LIN {X 0,Y 162.399,Z 558.631,A -85,B 0,C 180,E1 -26128.349,E2 -26128.349} C_VEL
LIN {X 0,Y 156.579,Z 567.786,A -85,B 0,C 180,E1 -26130.23,E2 -26130.23} C_VEL
LIN {X 0,Y 150.044,Z 576.728,A -85,B 0,C 180,E1 -26132.532,E2 -26132.532} C_VEL
LIN {X 0,Y 142.728,Z 585.711,A -85,B 0,C 180,E1 -26135.664,E2 -26135.664} C_VEL
LIN {X 0,Y 135.887,Z 593.161,A -85,B 0,C 180,E1 -26139.125,E2 -26139.125} C_VEL
LIN {X 0,Y 129.545,Z 599.346,A -85,B 0,C 180,E1 -26142.914,E2 -26142.914} C_VEL
LIN {X 0,Y 123.734,Z 604.443,A -85,B 0,C 180,E1 -26147.033,E2 -26147.033} C_VEL
LIN {X 0,Y 117.104,Z 609.682,A -85,B 0,C 180,E1 -26153.121,E2 -26153.121} C_VEL
LIN {X 0,Y 111.791,Z 613.372,A -85,B 0,C 180,E1 -26159.806,E2 -26159.806} C_VEL
LIN {X 0,Y 108.032,Z 615.635,A -85,B 0,C 180,E1 -26167.026,E2 -26167.026} C_VEL
LIN {X 0,Y 105.706,Z 616.545,A -85,B 0,C 180,E1 -26174.577,E2 -26174.577} C_VEL
LIN {X 0,Y 105.009,Z 616.121,A -85,B 0,C 180,E1 -26182.308,E2 -26182.308} C_VEL
LIN {X 0,Y 105.077,Z 615.416,A -85,B 0,C 180,E1 -26186.165,E2 -26186.165} C_VEL
LIN {X 0,Y 105.791,Z 613.021,A -85,B 0,C 180,E1 -26193.809,E2 -26193.809} C_VEL
LIN {X 0,Y 107.768,Z 609.248,A -85,B 0,C 180,E1 -26201.282,E2 -26201.282} C_VEL
LIN {X 0,Y 111.163,Z 603.939,A -85,B 0,C 180,E1 -26208.427,E2 -26208.427} C_VEL
LIN {X 0,Y 114.818,Z 598.843,A -85,B 0,C 180,E1 -26213.444,E2 -26213.444} C_VEL
LIN {X 0,Y 119.854,Z 591.564,A -85,B 0,C 180,E1 -26218.931,E2 -26218.931} C_VEL
LIN {X 0,Y 124.817,Z 583.942,A -85,B 0,C 180,E1 -26223.297,E2 -26223.297} C_VEL
LIN {X 0,Y 130.491,Z 574.792,A -85,B 0,C 180,E1 -26227.292,E2 -26227.292} C_VEL
LIN {X 0,Y 136.215,Z 564.684,A -85,B 0,C 180,E1 -26230.645,E2 -26230.645} C_VEL
LIN {X 0,Y 141.727,Z 553.57,A -85,B 0,C 180,E1 -26233.473,E2 -26233.473} C_VEL
LIN {X 0,Y 146.852,Z 541.305,A -85,B 0,C 180,E1 -26235.877,E2 -26235.877} C_VEL
LIN {X 0,Y 151.111,Z 529.497,A -85,B 0,C 180,E1 -26237.587,E2 -26237.587} C_VEL
LIN {X 0,Y 154.843,Z 516.616,A -85,B 0,C 180,E1 -26238.986,E2 -26238.986} C_VEL
LIN {X 0,Y 157.814,Z 502.413,A -85,B 0,C 180,E1 -26240.126,E2 -26240.126} C_VEL
LIN {X 0,Y 159.807,Z 487.984,A -85,B 0,C 180,E1 -26240.867,E2 -26240.867} C_VEL
LIN {X 0,Y 163.436,Z 443.82,A -85,B 0,C 180,E1 -26242.428,E2 -26242.428} C_VEL
LIN {X 0,Y 159.128,Z 434.822,A -85,B 0,C 180,E1 -26245.539,E2 -26245.539} C_VEL
LIN {X 0,Y 155.155,Z 427.48,A -85,B 0,C 180,E1 -26248.763,E2 -26248.763} C_VEL
LIN {X 0,Y 151.706,Z 421.59,A -85,B 0,C 180,E1 -26251.973,E2 -26251.973} C_VEL
LIN {X 0,Y 149.783,Z 418.5,A -85,B 0,C 180,E1 -26253.994,E2 -26253.994} C_VEL
LIN {X 0,Y 147.754,Z 415.273,A -85,B 0,C 180,E1 -26256.389,E2 -26256.389} C_VEL
LIN {X 0,Y 145.207,Z 411.371,A -85,B 0,C 180,E1 -26259.939,E2 -26259.939} C_VEL
LIN {X 0,Y 142.875,Z 408.164,A -85,B 0,C 180,E1 -26264.073,E2 -26264.073} C_VEL
LIN {X 0,Y 142.203,Z 406.763,A -85,B 0,C 180,E1 -26265.692,E2 -26265.692} C_VEL
LIN {X 0,Y 139.978,Z 403.826,A -85,B 0,C 180,E1 -26274.958,E2 -26274.958} C_VEL
LIN {X 0,Y 140.014,Z 403.461,A -85,B 0,C 180,E1 -26278.561,E2 -26278.561} C_VEL
LIN {X 0,Y 140.342,Z 404.521,A -85,B 0,C 180,E1 -26281.793,E2 -26281.793} C_VEL
LIN {X 0,Y 142.46,Z 406.94,A -85,B 0,C 180,E1 -26288.51,E2 -26288.51} C_VEL
LIN {X 0,Y 144.47,Z 410.538,A -85,B 0,C 180,E1 -26292.555,E2 -26292.555} C_VEL
LIN {X 0,Y 145.741,Z 412.18,A -85,B 0,C 180,E1 -26294.508,E2 -26294.508} C_VEL
LIN {X 0,Y 148.649,Z 416.668,A -85,B 0,C 180,E1 -26298.342,E2 -26298.342} C_VEL
LIN {X 0,Y 151.312,Z 420.86,A -85,B 0,C 180,E1 -26301.258,E2 -26301.258} C_VEL
LIN {X 0,Y 154.67,Z 426.429,A -85,B 0,C 180,E1 -26304.431,E2 -26304.431} C_VEL
LIN {X 0,Y 157.563,Z 432.02,A -85,B 0,C 180,E1 -26306.891,E2 -26306.891} C_VEL
LIN {X 0,Y 161.424,Z 442.286,A -85,B 0,C 180,E1 -26310.022,E2 -26310.022} C_VEL
LIN {X 0,Y 163.244,Z 447.912,A -85,B 0,C 180,E1 -26311.422,E2 -26311.422} C_VEL
LIN {X 0,Y 159.088,Z 496.229,A -85,B 0,C 180,E1 -26313.076,E2 -26313.076} C_VEL
LIN {X 0,Y 156.838,Z 510.579,A -85,B 0,C 180,E1 -26313.863,E2 -26313.863} C_VEL
LIN {X 0,Y 153.433,Z 524.942,A -85,B 0,C 180,E1 -26315.041,E2 -26315.041} C_VEL
LIN {X 0,Y 149.545,Z 537.278,A -85,B 0,C 180,E1 -26316.411,E2 -26316.411} C_VEL
LIN {X 0,Y 144.563,Z 550.226,A -85,B 0,C 180,E1 -26318.381,E2 -26318.381} C_VEL
LIN {X 0,Y 139.278,Z 561.994,A -85,B 0,C 180,E1 -26320.81,E2 -26320.81} C_VEL
LIN {X 0,Y 133.684,Z 572.756,A -85,B 0,C 180,E1 -26323.711,E2 -26323.711} C_VEL
LIN {X 0,Y 127.43,Z 583.411,A -85,B 0,C 180,E1 -26327.5,E2 -26327.5} C_VEL
LIN {X 0,Y 121.787,Z 592.198,A -85,B 0,C 180,E1 -26331.659,E2 -26331.659} C_VEL
LIN {X 0,Y 116.209,Z 600.631,A -85,B 0,C 180,E1 -26337.025,E2 -26337.025} C_VEL
LIN {X 0,Y 112.275,Z 606.497,A -85,B 0,C 180,E1 -26342.001,E2 -26342.001} C_VEL
LIN {X 0,Y 109.209,Z 611.326,A -85,B 0,C 180,E1 -26347.287,E2 -26347.287} C_VEL
LIN {X 0,Y 106.398,Z 616.311,A -85,B 0,C 180,E1 -26354.68,E2 -26354.68} C_VEL
LIN {X 0,Y 105.166,Z 619.78,A -85,B 0,C 180,E1 -26362.319,E2 -26362.319} C_VEL
LIN {X 0,Y 105.166,Z 621.827,A -85,B 0,C 180,E1 -26370,E2 -26370} C_VEL
LIN {X 0,Y 105.195,Z 622.477,A -85,B 0,C 180,E1 -26377.679,E2 -26377.679} C_VEL
LIN {X 0,Y 106.498,Z 621.795,A -85,B 0,C 180,E1 -26385.305,E2 -26385.305} C_VEL
LIN {X 0,Y 109.463,Z 619.789,A -85,B 0,C 180,E1 -26392.657,E2 -26392.657} C_VEL
LIN {X 0,Y 114.037,Z 616.407,A -85,B 0,C 180,E1 -26399.539,E2 -26399.539} C_VEL
LIN {X 0,Y 118.372,Z 612.921,A -85,B 0,C 180,E1 -26404.334,E2 -26404.334} C_VEL
LIN {X 0,Y 121.014,Z 610.729,A -85,B 0,C 180,E1 -26406.692,E2 -26406.692} C_VEL
LIN {X 0,Y 123.209,Z 608.466,A -85,B 0,C 180,E1 -26409.042,E2 -26409.042} C_VEL
LIN {X 0,Y 125.615,Z 604.474,A -85,B 0,C 180,E1 -26413.085,E2 -26413.085} C_VEL
LIN {X 0,Y 128.462,Z 599.904,A -85,B 0,C 180,E1 -26416.838,E2 -26416.838} C_VEL
LIN {X 0,Y 131.222,Z 596.74,A -85,B 0,C 180,E1 -26418.667,E2 -26418.667} C_VEL
LIN {X 0,Y 139.696,Z 587.753,A -85,B 0,C 180,E1 -26422.406,E2 -26422.406} C_VEL
LIN {X 0,Y 147.43,Z 578.268,A -85,B 0,C 180,E1 -26425.314,E2 -26425.314} C_VEL
LIN {X 0,Y 154.898,Z 567.778,A -85,B 0,C 180,E1 -26427.675,E2 -26427.675} C_VEL
LIN {X 0,Y 161.912,Z 556.21,A -85,B 0,C 180,E1 -26429.618,E2 -26429.618} C_VEL
LIN {X 0,Y 168.417,Z 543.379,A -85,B 0,C 180,E1 -26431.199,E2 -26431.199} C_VEL
LIN {X 0,Y 173.581,Z 530.831,A -85,B 0,C 180,E1 -26432.332,E2 -26432.332} C_VEL
LIN {X 0,Y 177.858,Z 517.413,A -85,B 0,C 180,E1 -26433.247,E2 -26433.247} C_VEL
LIN {X 0,Y 181.081,Z 503.535,A -85,B 0,C 180,E1 -26433.906,E2 -26433.906} C_VEL
LIN {X 0,Y 183.19,Z 488.883,A -85,B 0,C 180,E1 -26434.353,E2 -26434.353} C_VEL
LIN {X 0,Y 184.85,Z 471.444,A -85,B 0,C 180,E1 -26434.848,E2 -26434.848} C_VEL
LIN {X 0,Y 182.027,Z 462.8,A -85,B 0,C 180,E1 -26438.096,E2 -26438.096} C_VEL
LIN {X 0,Y 179.629,Z 456.499,A -85,B 0,C 180,E1 -26441.299,E2 -26441.299} C_VEL
LIN {X 0,Y 177.45,Z 452.505,A -85,B 0,C 180,E1 -26444.685,E2 -26444.685} C_VEL
LIN {X 0,Y 175.833,Z 449.251,A -85,B 0,C 180,E1 -26448.107,E2 -26448.107} C_VEL
LIN {X 0,Y 174.341,Z 445.787,A -85,B 0,C 180,E1 -26453.782,E2 -26453.782} C_VEL
LIN {X 0,Y 174.27,Z 445.225,A -85,B 0,C 180,E1 -26454.656,E2 -26454.656} C_VEL
LIN {X 0,Y 174.337,Z 445.109,A -85,B 0,C 180,E1 -26460.145,E2 -26460.145} C_VEL
LIN {X 0,Y 175.732,Z 448.882,A -85,B 0,C 180,E1 -26466.027,E2 -26466.027} C_VEL
LIN {X 0,Y 176.557,Z 450.738,A -85,B 0,C 180,E1 -26468.009,E2 -26468.009} C_VEL
LIN {X 0,Y 178.07,Z 453.628,A -85,B 0,C 180,E1 -26470.806,E2 -26470.806} C_VEL
LIN {X 0,Y 180.172,Z 457.72,A -85,B 0,C 180,E1 -26473.896,E2 -26473.896} C_VEL
LIN {X 0,Y 182.541,Z 462.521,A -85,B 0,C 180,E1 -26476.766,E2 -26476.766} C_VEL
LIN {X 0,Y 185.162,Z 468.275,A -85,B 0,C 180,E1 -26479.506,E2 -26479.506} C_VEL
LIN {X 0,Y 182.433,Z 493.552,A -85,B 0,C 180,E1 -26480.188,E2 -26480.188} C_VEL
LIN {X 0,Y 179.908,Z 506.993,A -85,B 0,C 180,E1 -26480.783,E2 -26480.783} C_VEL
LIN {X 0,Y 176.286,Z 520.463,A -85,B 0,C 180,E1 -26481.662,E2 -26481.662} C_VEL
LIN {X 0,Y 171.504,Z 533.661,A -85,B 0,C 180,E1 -26482.781,E2 -26482.781} C_VEL
LIN {X 0,Y 165.72,Z 546.39,A -85,B 0,C 180,E1 -26484.25,E2 -26484.25} C_VEL
LIN {X 0,Y 159.25,Z 558.074,A -85,B 0,C 180,E1 -26486.026,E2 -26486.026} C_VEL
LIN {X 0,Y 153.016,Z 567.649,A -85,B 0,C 180,E1 -26487.923,E2 -26487.923} C_VEL
LIN {X 0,Y 146.289,Z 576.569,A -85,B 0,C 180,E1 -26490.148,E2 -26490.148} C_VEL
LIN {X 0,Y 138.639,Z 585.613,A -85,B 0,C 180,E1 -26493.237,E2 -26493.237} C_VEL
LIN {X 0,Y 131.447,Z 593.117,A -85,B 0,C 180,E1 -26496.681,E2 -26496.681} C_VEL
LIN {X 0,Y 124.728,Z 599.348,A -85,B 0,C 180,E1 -26500.478,E2 -26500.478} C_VEL
LIN {X 0,Y 118.558,Z 604.472,A -85,B 0,C 180,E1 -26504.657,E2 -26504.657} C_VEL
LIN {X 0,Y 113.05,Z 608.576,A -85,B 0,C 180,E1 -26509.252,E2 -26509.252} C_VEL
LIN {X 0,Y 108.302,Z 611.817,A -85,B 0,C 180,E1 -26514.266,E2 -26514.266} C_VEL
LIN {X 0,Y 103.348,Z 614.818,A -85,B 0,C 180,E1 -26521.575,E2 -26521.575} C_VEL
LIN {X 0,Y 99.921,Z 616.434,A -85,B 0,C 180,E1 -26529.411,E2 -26529.411} C_VEL
LIN {X 0,Y 98.157,Z 616.711,A -85,B 0,C 180,E1 -26537.597,E2 -26537.597} C_VEL
LIN {X 0,Y 97.916,Z 616.351,A -85,B 0,C 180,E1 -26541.747,E2 -26541.747} C_VEL
LIN {X 0,Y 97.955,Z 615.663,A -85,B 0,C 180,E1 -26545.886,E2 -26545.886} C_VEL
LIN {X 0,Y 98.489,Z 613.862,A -85,B 0,C 180,E1 -26552.507,E2 -26552.507} C_VEL
LIN {X 0,Y 100.145,Z 610.623,A -85,B 0,C 180,E1 -26560.104,E2 -26560.104} C_VEL
LIN {X 0,Y 103.446,Z 605.748,A -85,B 0,C 180,E1 -26567.801,E2 -26567.801} C_VEL
LIN {X 0,Y 108.372,Z 599.241,A -85,B 0,C 180,E1 -26574.93,E2 -26574.93} C_VEL
LIN {X 0,Y 113.705,Z 592.01,A -85,B 0,C 180,E1 -26580.658,E2 -26580.658} C_VEL
LIN {X 0,Y 119.932,Z 583.053,A -85,B 0,C 180,E1 -26585.872,E2 -26585.872} C_VEL
LIN {X 0,Y 126.016,Z 573.655,A -85,B 0,C 180,E1 -26589.892,E2 -26589.892} C_VEL
LIN {X 0,Y 132.065,Z 563.253,A -85,B 0,C 180,E1 -26593.246,E2 -26593.246} C_VEL
LIN {X 0,Y 137.885,Z 551.772,A -85,B 0,C 180,E1 -26596.049,E2 -26596.049} C_VEL
LIN {X 0,Y 143.246,Z 539.058,A -85,B 0,C 180,E1 -26598.433,E2 -26598.433} C_VEL
LIN {X 0,Y 147.711,Z 526.619,A -85,B 0,C 180,E1 -26600.103,E2 -26600.103} C_VEL
LIN {X 0,Y 151.593,Z 512.787,A -85,B 0,C 180,E1 -26601.473,E2 -26601.473} C_VEL
LIN {X 0,Y 154.383,Z 498.867,A -85,B 0,C 180,E1 -26602.453,E2 -26602.453} C_VEL
LIN {X 0,Y 156.03,Z 485.645,A -85,B 0,C 180,E1 -26603.065,E2 -26603.065} C_VEL
LIN {X 0,Y 159.29,Z 446.776,A -85,B 0,C 180,E1 -26604.439,E2 -26604.439} C_VEL
LIN {X 0,Y 155.497,Z 438.74,A -85,B 0,C 180,E1 -26607.464,E2 -26607.464} C_VEL
LIN {X 0,Y 151.515,Z 431.095,A -85,B 0,C 180,E1 -26611.088,E2 -26611.088} C_VEL
LIN {X 0,Y 147.933,Z 424.893,A -85,B 0,C 180,E1 -26614.934,E2 -26614.934} C_VEL
LIN {X 0,Y 145.849,Z 421.5,A -85,B 0,C 180,E1 -26617.575,E2 -26617.575} C_VEL
LIN {X 0,Y 143.612,Z 417.914,A -85,B 0,C 180,E1 -26620.965,E2 -26620.965} C_VEL
LIN {X 0,Y 141.494,Z 414.599,A -85,B 0,C 180,E1 -26625.141,E2 -26625.141} C_VEL
LIN {X 0,Y 140.971,Z 413.609,A -85,B 0,C 180,E1 -26626.496,E2 -26626.496} C_VEL
LIN {X 0,Y 139.081,Z 410.76,A -85,B 0,C 180,E1 -26635.652,E2 -26635.652} C_VEL
LIN {X 0,Y 139.161,Z 410.509,A -85,B 0,C 180,E1 -26638.748,E2 -26638.748} C_VEL
LIN {X 0,Y 141.212,Z 413.663,A -85,B 0,C 180,E1 -26647.686,E2 -26647.686} C_VEL
LIN {X 0,Y 143.208,Z 417.38,A -85,B 0,C 180,E1 -26651.993,E2 -26651.993} C_VEL
LIN {X 0,Y 144.165,Z 418.711,A -85,B 0,C 180,E1 -26653.568,E2 -26653.568} C_VEL
LIN {X 0,Y 146.863,Z 423.102,A -85,B 0,C 180,E1 -26657.391,E2 -26657.391} C_VEL
LIN {X 0,Y 149.334,Z 427.228,A -85,B 0,C 180,E1 -26660.29,E2 -26660.29} C_VEL
LIN {X 0,Y 152.413,Z 432.646,A -85,B 0,C 180,E1 -26663.406,E2 -26663.406} C_VEL
LIN {X 0,Y 154.808,Z 437.586,A -85,B 0,C 180,E1 -26665.604,E2 -26665.604} C_VEL
LIN {X 0,Y 158.029,Z 446.818,A -85,B 0,C 180,E1 -26668.469,E2 -26668.469} C_VEL
LIN {X 0,Y 159.119,Z 450.292,A -85,B 0,C 180,E1 -26669.391,E2 -26669.391} C_VEL
LIN {X 0,Y 154.956,Z 496.665,A -85,B 0,C 180,E1 -26670.977,E2 -26670.977} C_VEL
LIN {X 0,Y 152.432,Z 511.607,A -85,B 0,C 180,E1 -26671.815,E2 -26671.815} C_VEL
LIN {X 0,Y 148.784,Z 526.107,A -85,B 0,C 180,E1 -26673.027,E2 -26673.027} C_VEL
LIN {X 0,Y 144.108,Z 539.922,A -85,B 0,C 180,E1 -26674.619,E2 -26674.619} C_VEL
LIN {X 0,Y 138.978,Z 552.325,A -85,B 0,C 180,E1 -26676.605,E2 -26676.605} C_VEL
LIN {X 0,Y 133.194,Z 564.32,A -85,B 0,C 180,E1 -26679.22,E2 -26679.22} C_VEL
LIN {X 0,Y 127.695,Z 574.128,A -85,B 0,C 180,E1 -26682.014,E2 -26682.014} C_VEL
LIN {X 0,Y 121.2,Z 584.505,A -85,B 0,C 180,E1 -26685.907,E2 -26685.907} C_VEL
LIN {X 0,Y 115.329,Z 593.074,A -85,B 0,C 180,E1 -26690.221,E2 -26690.221} C_VEL
LIN {X 0,Y 109.496,Z 601.257,A -85,B 0,C 180,E1 -26695.833,E2 -26695.833} C_VEL
LIN {X 0,Y 104.785,Z 607.85,A -85,B 0,C 180,E1 -26701.999,E2 -26701.999} C_VEL
LIN {X 0,Y 101.703,Z 612.419,A -85,B 0,C 180,E1 -26707.663,E2 -26707.663} C_VEL
LIN {X 0,Y 99.513,Z 616.001,A -85,B 0,C 180,E1 -26713.591,E2 -26713.591} C_VEL
LIN {X 0,Y 98.102,Z 619.505,A -85,B 0,C 180,E1 -26721.763,E2 -26721.763} C_VEL
LIN {X 0,Y 98.072,Z 621.586,A -85,B 0,C 180,E1 -26730,E2 -26730} C_VEL
LIN {X 0,Y 98.129,Z 622.268,A -85,B 0,C 180,E1 -26738.235,E2 -26738.235} C_VEL
LIN {X 0,Y 99.633,Z 621.623,A -85,B 0,C 180,E1 -26746.388,E2 -26746.388} C_VEL
LIN {X 0,Y 102.905,Z 619.655,A -85,B 0,C 180,E1 -26754.19,E2 -26754.19} C_VEL
LIN {X 0,Y 107.866,Z 616.311,A -85,B 0,C 180,E1 -26761.414,E2 -26761.414} C_VEL
LIN {X 0,Y 114.305,Z 611.496,A -85,B 0,C 180,E1 -26767.939,E2 -26767.939} C_VEL
LIN {X 0,Y 122.175,Z 605.076,A -85,B 0,C 180,E1 -26773.652,E2 -26773.652} C_VEL
LIN {X 0,Y 129.941,Z 597.954,A -85,B 0,C 180,E1 -26778.045,E2 -26778.045} C_VEL
LIN {X 0,Y 131.222,Z 596.74,A -85,B 0,C 180,E1 -26778.667,E2 -26778.667} C_VEL
LIN {X 0,Y 134.055,Z 593.448,A -85,B 0,C 180,E1 -26780.395,E2 -26780.395} C_VEL
LIN {X 0,Y 137.498,Z 587.894,A -85,B 0,C 180,E1 -26783.565,E2 -26783.565} C_VEL
LIN {X 0,Y 141.049,Z 581.916,A -85,B 0,C 180,E1 -26786.479,E2 -26786.479} C_VEL
LIN {X 0,Y 143.92,Z 577.893,A -85,B 0,C 180,E1 -26787.779,E2 -26787.779} C_VEL
LIN {X 0,Y 151.944,Z 566.941,A -85,B 0,C 180,E1 -26790.139,E2 -26790.139} C_VEL
LIN {X 0,Y 158.448,Z 556.531,A -85,B 0,C 180,E1 -26791.829,E2 -26791.829} C_VEL
LIN {X 0,Y 165.122,Z 543.818,A -85,B 0,C 180,E1 -26793.353,E2 -26793.353} C_VEL
LIN {X 0,Y 170.41,Z 531.434,A -85,B 0,C 180,E1 -26794.44,E2 -26794.44} C_VEL
LIN {X 0,Y 175.109,Z 517.206,A -85,B 0,C 180,E1 -26795.37,E2 -26795.37} C_VEL
LIN {X 0,Y 178.509,Z 502.772,A -85,B 0,C 180,E1 -26796.029,E2 -26796.029} C_VEL
LIN {X 0,Y 180.553,Z 488.752,A -85,B 0,C 180,E1 -26796.43,E2 -26796.43} C_VEL
LIN {X 0,Y 181.92,Z 474.663,A -85,B 0,C 180,E1 -26796.836,E2 -26796.836} C_VEL
LIN {X 0,Y 179.482,Z 466.859,A -85,B 0,C 180,E1 -26800.035,E2 -26800.035} C_VEL
LIN {X 0,Y 177.95,Z 462.707,A -85,B 0,C 180,E1 -26802.326,E2 -26802.326} C_VEL
LIN {X 0,Y 176.126,Z 459.105,A -85,B 0,C 180,E1 -26805.426,E2 -26805.426} C_VEL
LIN {X 0,Y 174.721,Z 456.052,A -85,B 0,C 180,E1 -26808.662,E2 -26808.662} C_VEL
LIN {X 0,Y 173.424,Z 452.799,A -85,B 0,C 180,E1 -26814.088,E2 -26814.088} C_VEL
LIN {X 0,Y 173.326,Z 452.222,A -85,B 0,C 180,E1 -26815.349,E2 -26815.349} C_VEL
LIN {X 0,Y 173.429,Z 452.11,A -85,B 0,C 180,E1 -26819.829,E2 -26819.829} C_VEL
LIN {X 0,Y 175.004,Z 456.528,A -85,B 0,C 180,E1 -26826.486,E2 -26826.486} C_VEL
LIN {X 0,Y 176.777,Z 460.397,A -85,B 0,C 180,E1 -26830.208,E2 -26830.208} C_VEL
LIN {X 0,Y 178.843,Z 464.644,A -85,B 0,C 180,E1 -26833.421,E2 -26833.421} C_VEL
LIN {X 0,Y 181.419,Z 470.314,A -85,B 0,C 180,E1 -26836.674,E2 -26836.674} C_VEL
LIN {X 0,Y 182.18,Z 472.157,A -85,B 0,C 180,E1 -26837.542,E2 -26837.542} C_VEL
LIN {X 0,Y 179.568,Z 494.782,A -85,B 0,C 180,E1 -26838.137,E2 -26838.137} C_VEL
LIN {X 0,Y 176.769,Z 508.76,A -85,B 0,C 180,E1 -26838.764,E2 -26838.764} C_VEL
LIN {X 0,Y 172.935,Z 522.183,A -85,B 0,C 180,E1 -26839.644,E2 -26839.644} C_VEL
LIN {X 0,Y 168.103,Z 534.871,A -85,B 0,C 180,E1 -26840.703,E2 -26840.703} C_VEL
LIN {X 0,Y 162.162,Z 547.405,A -85,B 0,C 180,E1 -26842.126,E2 -26842.126} C_VEL
LIN {X 0,Y 155.581,Z 558.823,A -85,B 0,C 180,E1 -26843.834,E2 -26843.834} C_VEL
LIN {X 0,Y 149.638,Z 567.613,A -85,B 0,C 180,E1 -26845.526,E2 -26845.526} C_VEL
LIN {X 0,Y 141.449,Z 578.052,A -85,B 0,C 180,E1 -26848.128,E2 -26848.128} C_VEL
LIN {X 0,Y 133.521,Z 586.878,A -85,B 0,C 180,E1 -26851.206,E2 -26851.206} C_VEL
LIN {X 0,Y 124.851,Z 595.313,A -85,B 0,C 180,E1 -26855.294,E2 -26855.294} C_VEL
LIN {X 0,Y 117.917,Z 601.164,A -85,B 0,C 180,E1 -26859.214,E2 -26859.214} C_VEL
LIN {X 0,Y 110.31,Z 606.836,A -85,B 0,C 180,E1 -26864.495,E2 -26864.495} C_VEL
LIN {X 0,Y 104.162,Z 610.916,A -85,B 0,C 180,E1 -26870.136,E2 -26870.136} C_VEL
LIN {X 0,Y 99.562,Z 613.62,A -85,B 0,C 180,E1 -26875.619,E2 -26875.619} C_VEL
LIN {X 0,Y 94.955,Z 615.955,A -85,B 0,C 180,E1 -26883.636,E2 -26883.636} C_VEL
LIN {X 0,Y 91.918,Z 616.935,A -85,B 0,C 180,E1 -26892.192,E2 -26892.192} C_VEL
LIN {X 0,Y 90.825,Z 616.581,A -85,B 0,C 180,E1 -26901.097,E2 -26901.097} C_VEL
LIN {X 0,Y 90.832,Z 615.91,A -85,B 0,C 180,E1 -26905.562,E2 -26905.562} C_VEL
LIN {X 0,Y 91.58,Z 613.745,A -85,B 0,C 180,E1 -26913.906,E2 -26913.906} C_VEL
LIN {X 0,Y 93.181,Z 610.941,A -85,B 0,C 180,E1 -26920.868,E2 -26920.868} C_VEL
LIN {X 0,Y 96.728,Z 606.104,A -85,B 0,C 180,E1 -26929.086,E2 -26929.086} C_VEL
LIN {X 0,Y 102.006,Z 599.639,A -85,B 0,C 180,E1 -26936.604,E2 -26936.604} C_VEL
LIN {X 0,Y 107.689,Z 592.454,A -85,B 0,C 180,E1 -26942.574,E2 -26942.574} C_VEL
LIN {X 0,Y 113.271,Z 584.935,A -85,B 0,C 180,E1 -26947.224,E2 -26947.224} C_VEL
LIN {X 0,Y 119.561,Z 575.904,A -85,B 0,C 180,E1 -26951.397,E2 -26951.397} C_VEL
LIN {X 0,Y 126.424,Z 564.966,A -85,B 0,C 180,E1 -26955.134,E2 -26955.134} C_VEL
LIN {X 0,Y 132.465,Z 553.819,A -85,B 0,C 180,E1 -26957.967,E2 -26957.967} C_VEL
LIN {X 0,Y 138.056,Z 541.514,A -85,B 0,C 180,E1 -26960.349,E2 -26960.349} C_VEL
LIN {X 0,Y 142.636,Z 529.661,A -85,B 0,C 180,E1 -26962.03,E2 -26962.03} C_VEL
LIN {X 0,Y 146.655,Z 516.703,A -85,B 0,C 180,E1 -26963.386,E2 -26963.386} C_VEL
LIN {X 0,Y 149.768,Z 502.759,A -85,B 0,C 180,E1 -26964.483,E2 -26964.483} C_VEL
LIN {X 0,Y 151.886,Z 488.576,A -85,B 0,C 180,E1 -26965.188,E2 -26965.188} C_VEL
LIN {X 0,Y 155.349,Z 449.891,A -85,B 0,C 180,E1 -26966.539,E2 -26966.539} C_VEL
LIN {X 0,Y 151.516,Z 441.574,A -85,B 0,C 180,E1 -26969.983,E2 -26969.983} C_VEL
LIN {X 0,Y 147.819,Z 434.344,A -85,B 0,C 180,E1 -26973.856,E2 -26973.856} C_VEL
LIN {X 0,Y 144.657,Z 428.574,A -85,B 0,C 180,E1 -26977.886,E2 -26977.886} C_VEL
LIN {X 0,Y 142.201,Z 424.617,A -85,B 0,C 180,E1 -26981.773,E2 -26981.773} C_VEL
LIN {X 0,Y 140.176,Z 421.09,A -85,B 0,C 180,E1 -26986.184,E2 -26986.184} C_VEL
LIN {X 0,Y 139.77,Z 420.435,A -85,B 0,C 180,E1 -26987.314,E2 -26987.314} C_VEL
LIN {X 0,Y 138.213,Z 417.825,A -85,B 0,C 180,E1 -26995.625,E2 -26995.625} C_VEL
LIN {X 0,Y 138.29,Z 417.586,A -85,B 0,C 180,E1 -26998.74,E2 -26998.74} C_VEL
LIN {X 0,Y 139.76,Z 420.171,A -85,B 0,C 180,E1 -27006.224,E2 -27006.224} C_VEL
LIN {X 0,Y 140.228,Z 421.048,A -85,B 0,C 180,E1 -27007.559,E2 -27007.559} C_VEL
LIN {X 0,Y 142.79,Z 425.525,A -85,B 0,C 180,E1 -27012.886,E2 -27012.886} C_VEL
LIN {X 0,Y 145.194,Z 429.676,A -85,B 0,C 180,E1 -27016.521,E2 -27016.521} C_VEL
LIN {X 0,Y 147.838,Z 434.334,A -85,B 0,C 180,E1 -27019.798,E2 -27019.798} C_VEL
LIN {X 0,Y 151.108,Z 440.678,A -85,B 0,C 180,E1 -27023.252,E2 -27023.252} C_VEL
LIN {X 0,Y 152.63,Z 444.656,A -85,B 0,C 180,E1 -27024.779,E2 -27024.779} C_VEL
LIN {X 0,Y 155.224,Z 452.859,A -85,B 0,C 180,E1 -27027.284,E2 -27027.284} C_VEL
LIN {X 0,Y 151.135,Z 496.354,A -85,B 0,C 180,E1 -27028.736,E2 -27028.736} C_VEL
LIN {X 0,Y 148.706,Z 510.587,A -85,B 0,C 180,E1 -27029.51,E2 -27029.51} C_VEL
LIN {X 0,Y 145.357,Z 523.857,A -85,B 0,C 180,E1 -27030.548,E2 -27030.548} C_VEL
LIN {X 0,Y 140.861,Z 537.233,A -85,B 0,C 180,E1 -27031.988,E2 -27031.988} C_VEL
LIN {X 0,Y 135.473,Z 550.107,A -85,B 0,C 180,E1 -27033.9,E2 -27033.9} C_VEL
LIN {X 0,Y 129.439,Z 562.407,A -85,B 0,C 180,E1 -27036.457,E2 -27036.457} C_VEL
LIN {X 0,Y 123.04,Z 573.535,A -85,B 0,C 180,E1 -27039.548,E2 -27039.548} C_VEL
LIN {X 0,Y 116.163,Z 583.989,A -85,B 0,C 180,E1 -27043.449,E2 -27043.449} C_VEL
LIN {X 0,Y 109.913,Z 592.611,A -85,B 0,C 180,E1 -27047.828,E2 -27047.828} C_VEL
LIN {X 0,Y 103.637,Z 600.85,A -85,B 0,C 180,E1 -27053.605,E2 -27053.605} C_VEL
LIN {X 0,Y 98.518,Z 607.484,A -85,B 0,C 180,E1 -27060.043,E2 -27060.043} C_VEL
LIN {X 0,Y 95.139,Z 612.077,A -85,B 0,C 180,E1 -27066.029,E2 -27066.029} C_VEL
LIN {X 0,Y 92.676,Z 615.692,A -85,B 0,C 180,E1 -27072.343,E2 -27072.343} C_VEL
LIN {X 0,Y 91.065,Z 619.231,A -85,B 0,C 180,E1 -27081.121,E2 -27081.121} C_VEL
LIN {X 0,Y 90.97,Z 621.345,A -85,B 0,C 180,E1 -27090,E2 -27090} C_VEL
LIN {X 0,Y 91.091,Z 622.057,A -85,B 0,C 180,E1 -27098.876,E2 -27098.876} C_VEL
LIN {X 0,Y 92.817,Z 621.446,A -85,B 0,C 180,E1 -27107.63,E2 -27107.63} C_VEL
LIN {X 0,Y 96.434,Z 619.517,A -85,B 0,C 180,E1 -27115.929,E2 -27115.929} C_VEL
LIN {X 0,Y 101.817,Z 616.214,A -85,B 0,C 180,E1 -27123.518,E2 -27123.518} C_VEL
LIN {X 0,Y 108.759,Z 611.436,A -85,B 0,C 180,E1 -27130.254,E2 -27130.254} C_VEL
LIN {X 0,Y 117.115,Z 605.054,A -85,B 0,C 180,E1 -27136.062,E2 -27136.062} C_VEL
LIN {X 0,Y 125.302,Z 597.975,A -85,B 0,C 180,E1 -27140.462,E2 -27140.462} C_VEL
LIN {X 0,Y 134.175,Z 589.236,A -85,B 0,C 180,E1 -27144.278,E2 -27144.278} C_VEL
LIN {X 0,Y 142.148,Z 580.112,A -85,B 0,C 180,E1 -27147.191,E2 -27147.191} C_VEL
LIN {X 0,Y 143.92,Z 577.893,A -85,B 0,C 180,E1 -27147.779,E2 -27147.779} C_VEL
LIN {X 0,Y 146.8,Z 573.767,A -85,B 0,C 180,E1 -27148.979,E2 -27148.979} C_VEL
LIN {X 0,Y 150.415,Z 566.827,A -85,B 0,C 180,E1 -27151.317,E2 -27151.317} C_VEL
LIN {X 0,Y 153.904,Z 559.577,A -85,B 0,C 180,E1 -27153.479,E2 -27153.479} C_VEL
LIN {X 0,Y 156.442,Z 554.807,A -85,B 0,C 180,E1 -27154.39,E2 -27154.39} C_VEL
LIN {X 0,Y 162.84,Z 542.68,A -85,B 0,C 180,E1 -27155.742,E2 -27155.742} C_VEL
LIN {X 0,Y 168.275,Z 530.052,A -85,B 0,C 180,E1 -27156.752,E2 -27156.752} C_VEL
LIN {X 0,Y 172.588,Z 517.052,A -85,B 0,C 180,E1 -27157.558,E2 -27157.558} C_VEL
LIN {X 0,Y 175.928,Z 503.282,A -85,B 0,C 180,E1 -27158.161,E2 -27158.161} C_VEL
LIN {X 0,Y 178.171,Z 488.502,A -85,B 0,C 180,E1 -27158.57,E2 -27158.57} C_VEL
LIN {X 0,Y 179.189,Z 478.059,A -85,B 0,C 180,E1 -27158.891,E2 -27158.891} C_VEL
LIN {X 0,Y 177.432,Z 472.101,A -85,B 0,C 180,E1 -27161.527,E2 -27161.527} C_VEL
LIN {X 0,Y 176.375,Z 469.014,A -85,B 0,C 180,E1 -27163.298,E2 -27163.298} C_VEL
LIN {X 0,Y 174.822,Z 465.713,A -85,B 0,C 180,E1 -27166.191,E2 -27166.191} C_VEL
LIN {X 0,Y 173.583,Z 462.815,A -85,B 0,C 180,E1 -27169.34,E2 -27169.34} C_VEL
LIN {X 0,Y 172.492,Z 459.535,A -85,B 0,C 180,E1 -27174.782,E2 -27174.782} C_VEL
LIN {X 0,Y 172.504,Z 459.099,A -85,B 0,C 180,E1 -27179.31,E2 -27179.31} C_VEL
LIN {X 0,Y 173.866,Z 463.3,A -85,B 0,C 180,E1 -27185.873,E2 -27185.873} C_VEL
LIN {X 0,Y 175.429,Z 466.975,A -85,B 0,C 180,E1 -27189.455,E2 -27189.455} C_VEL
LIN {X 0,Y 177.576,Z 471.665,A -85,B 0,C 180,E1 -27193.009,E2 -27193.009} C_VEL
LIN {X 0,Y 179.384,Z 476.043,A -85,B 0,C 180,E1 -27195.481,E2 -27195.481} C_VEL
LIN {X 0,Y 177.041,Z 495.503,A -85,B 0,C 180,E1 -27196.02,E2 -27196.02} C_VEL
LIN {X 0,Y 174.065,Z 509.733,A -85,B 0,C 180,E1 -27196.644,E2 -27196.644} C_VEL
LIN {X 0,Y 170.209,Z 522.731,A -85,B 0,C 180,E1 -27197.472,E2 -27197.472} C_VEL
LIN {X 0,Y 164.935,Z 536.082,A -85,B 0,C 180,E1 -27198.547,E2 -27198.547} C_VEL
LIN {X 0,Y 158.835,Z 548.42,A -85,B 0,C 180,E1 -27199.911,E2 -27199.911} C_VEL
LIN {X 0,Y 152.075,Z 559.694,A -85,B 0,C 180,E1 -27201.56,E2 -27201.56} C_VEL
LIN {X 0,Y 145.439,Z 569.07,A -85,B 0,C 180,E1 -27203.35,E2 -27203.35} C_VEL
LIN {X 0,Y 136.788,Z 579.535,A -85,B 0,C 180,E1 -27205.96,E2 -27205.96} C_VEL
LIN {X 0,Y 128.581,Z 588.144,A -85,B 0,C 180,E1 -27209.014,E2 -27209.014} C_VEL
LIN {X 0,Y 119.56,Z 596.341,A -85,B 0,C 180,E1 -27213.11,E2 -27213.11} C_VEL
LIN {X 0,Y 111.152,Z 602.909,A -85,B 0,C 180,E1 -27217.783,E2 -27217.783} C_VEL
LIN {X 0,Y 102.515,Z 608.709,A -85,B 0,C 180,E1 -27223.961,E2 -27223.961} C_VEL
LIN {X 0,Y 96.932,Z 612.028,A -85,B 0,C 180,E1 -27229.268,E2 -27229.268} C_VEL
LIN {X 0,Y 90.888,Z 615.103,A -85,B 0,C 180,E1 -27237.23,E2 -27237.23} C_VEL
LIN {X 0,Y 86.597,Z 616.789,A -85,B 0,C 180,E1 -27246.06,E2 -27246.06} C_VEL
LIN {X 0,Y 84.187,Z 617.136,A -85,B 0,C 180,E1 -27255.497,E2 -27255.497} C_VEL
LIN {X 0,Y 83.735,Z 616.156,A -85,B 0,C 180,E1 -27265.185,E2 -27265.185} C_VEL
LIN {X 0,Y 84.013,Z 615.175,A -85,B 0,C 180,E1 -27270,E2 -27270} C_VEL
LIN {X 0,Y 85.589,Z 612.209,A -85,B 0,C 180,E1 -27279.452,E2 -27279.452} C_VEL
LIN {X 0,Y 88.938,Z 607.82,A -85,B 0,C 180,E1 -27288.426,E2 -27288.426} C_VEL
LIN {X 0,Y 92.645,Z 603.467,A -85,B 0,C 180,E1 -27294.659,E2 -27294.659} C_VEL
LIN {X 0,Y 98.181,Z 597.162,A -85,B 0,C 180,E1 -27301.262,E2 -27301.262} C_VEL
LIN {X 0,Y 104.628,Z 589.338,A -85,B 0,C 180,E1 -27307.195,E2 -27307.195} C_VEL
LIN {X 0,Y 110.996,Z 581.151,A -85,B 0,C 180,E1 -27311.668,E2 -27311.668} C_VEL
LIN {X 0,Y 117.91,Z 571.294,A -85,B 0,C 180,E1 -27315.663,E2 -27315.663} C_VEL
LIN {X 0,Y 124.627,Z 560.343,A -85,B 0,C 180,E1 -27318.958,E2 -27318.958} C_VEL
LIN {X 0,Y 130.412,Z 549.454,A -85,B 0,C 180,E1 -27321.388,E2 -27321.388} C_VEL
LIN {X 0,Y 135.669,Z 537.688,A -85,B 0,C 180,E1 -27323.409,E2 -27323.409} C_VEL
LIN {X 0,Y 140.483,Z 524.783,A -85,B 0,C 180,E1 -27325.002,E2 -27325.002} C_VEL
LIN {X 0,Y 144.411,Z 510.837,A -85,B 0,C 180,E1 -27326.278,E2 -27326.278} C_VEL
LIN {X 0,Y 147.213,Z 496.711,A -85,B 0,C 180,E1 -27327.167,E2 -27327.167} C_VEL
LIN {X 0,Y 149.088,Z 481.099,A -85,B 0,C 180,E1 -27327.767,E2 -27327.767} C_VEL
LIN {X 0,Y 151.662,Z 453.196,A -85,B 0,C 180,E1 -27328.701,E2 -27328.701} C_VEL
LIN {X 0,Y 148.308,Z 445.742,A -85,B 0,C 180,E1 -27332.08,E2 -27332.08} C_VEL
LIN {X 0,Y 145.363,Z 439.695,A -85,B 0,C 180,E1 -27335.544,E2 -27335.544} C_VEL
LIN {X 0,Y 142.684,Z 434.584,A -85,B 0,C 180,E1 -27339.339,E2 -27339.339} C_VEL
LIN {X 0,Y 140.711,Z 431.121,A -85,B 0,C 180,E1 -27342.813,E2 -27342.813} C_VEL
LIN {X 0,Y 138.726,Z 427.36,A -85,B 0,C 180,E1 -27347.77,E2 -27347.77} C_VEL
LIN {X 0,Y 137.346,Z 424.894,A -85,B 0,C 180,E1 -27355.597,E2 -27355.597} C_VEL
LIN {X 0,Y 137.415,Z 424.686,A -85,B 0,C 180,E1 -27358.732,E2 -27358.732} C_VEL
LIN {X 0,Y 138.948,Z 427.552,A -85,B 0,C 180,E1 -27366.488,E2 -27366.488} C_VEL
LIN {X 0,Y 141.294,Z 432.074,A -85,B 0,C 180,E1 -27371.93,E2 -27371.93} C_VEL
LIN {X 0,Y 143.493,Z 436.12,A -85,B 0,C 180,E1 -27375.535,E2 -27375.535} C_VEL
LIN {X 0,Y 146.269,Z 441.301,A -85,B 0,C 180,E1 -27379.197,E2 -27379.197} C_VEL
LIN {X 0,Y 149.141,Z 447.563,A -85,B 0,C 180,E1 -27382.447,E2 -27382.447} C_VEL
LIN {X 0,Y 151.508,Z 455.364,A -85,B 0,C 180,E1 -27385.041,E2 -27385.041} C_VEL
LIN {X 0,Y 147.571,Z 495.994,A -85,B 0,C 180,E1 -27386.388,E2 -27386.388} C_VEL
LIN {X 0,Y 145.05,Z 510.308,A -85,B 0,C 180,E1 -27387.137,E2 -27387.137} C_VEL
LIN {X 0,Y 141.506,Z 523.878,A -85,B 0,C 180,E1 -27388.171,E2 -27388.171} C_VEL
LIN {X 0,Y 137.224,Z 536.32,A -85,B 0,C 180,E1 -27389.467,E2 -27389.467} C_VEL
LIN {X 0,Y 131.639,Z 549.332,A -85,B 0,C 180,E1 -27391.33,E2 -27391.33} C_VEL
LIN {X 0,Y 125.735,Z 560.989,A -85,B 0,C 180,E1 -27393.657,E2 -27393.657} C_VEL
LIN {X 0,Y 119.897,Z 570.974,A -85,B 0,C 180,E1 -27396.297,E2 -27396.297} C_VEL
LIN {X 0,Y 113.745,Z 580.179,A -85,B 0,C 180,E1 -27399.437,E2 -27399.437} C_VEL
LIN {X 0,Y 106.831,Z 589.4,A -85,B 0,C 180,E1 -27403.645,E2 -27403.645} C_VEL
LIN {X 0,Y 99.812,Z 598.222,A -85,B 0,C 180,E1 -27409.361,E2 -27409.361} C_VEL
LIN {X 0,Y 93.893,Z 605.211,A -85,B 0,C 180,E1 -27415.671,E2 -27415.671} C_VEL
LIN {X 0,Y 89.756,Z 610.286,A -85,B 0,C 180,E1 -27421.979,E2 -27421.979} C_VEL
LIN {X 0,Y 85.871,Z 615.381,A -85,B 0,C 180,E1 -27430.891,E2 -27430.891} C_VEL
LIN {X 0,Y 84.025,Z 618.955,A -85,B 0,C 180,E1 -27440.37,E2 -27440.37} C_VEL
LIN {X 0,Y 83.876,Z 621.103,A -85,B 0,C 180,E1 -27450,E2 -27450} C_VEL
LIN {X 0,Y 83.778,Z 621.643,A -85,B 0,C 180,E1 -27454.812,E2 -27454.812} C_VEL
LIN {X 0,Y 84.802,Z 621.721,A -85,B 0,C 180,E1 -27464.396,E2 -27464.396} C_VEL
LIN {X 0,Y 87.743,Z 620.484,A -85,B 0,C 180,E1 -27473.608,E2 -27473.608} C_VEL
LIN {X 0,Y 92.784,Z 617.92,A -85,B 0,C 180,E1 -27482.019,E2 -27482.019} C_VEL
LIN {X 0,Y 99.468,Z 613.938,A -85,B 0,C 180,E1 -27489.486,E2 -27489.486} C_VEL
LIN {X 0,Y 107.699,Z 608.417,A -85,B 0,C 180,E1 -27495.873,E2 -27495.873} C_VEL
LIN {X 0,Y 115.853,Z 602.211,A -85,B 0,C 180,E1 -27500.663,E2 -27500.663} C_VEL
LIN {X 0,Y 124.819,Z 594.495,A -85,B 0,C 180,E1 -27504.727,E2 -27504.727} C_VEL
LIN {X 0,Y 132.891,Z 586.465,A -85,B 0,C 180,E1 -27507.795,E2 -27507.795} C_VEL
LIN {X 0,Y 141.259,Z 576.807,A -85,B 0,C 180,E1 -27510.534,E2 -27510.534} C_VEL
LIN {X 0,Y 149.285,Z 566.105,A -85,B 0,C 180,E1 -27512.694,E2 -27512.694} C_VEL
LIN {X 0,Y 156.009,Z 555.562,A -85,B 0,C 180,E1 -27514.283,E2 -27514.283} C_VEL
LIN {X 0,Y 156.442,Z 554.807,A -85,B 0,C 180,E1 -27514.39,E2 -27514.39} C_VEL
LIN {X 0,Y 158.901,Z 549.951,A -85,B 0,C 180,E1 -27515.237,E2 -27515.237} C_VEL
LIN {X 0,Y 161.973,Z 541.917,A -85,B 0,C 180,E1 -27517.004,E2 -27517.004} C_VEL
LIN {X 0,Y 164.71,Z 533.566,A -85,B 0,C 180,E1 -27518.592,E2 -27518.592} C_VEL
LIN {X 0,Y 166.561,Z 528.22,A -85,B 0,C 180,E1 -27519.164,E2 -27519.164} C_VEL
LIN {X 0,Y 170.987,Z 514.668,A -85,B 0,C 180,E1 -27519.903,E2 -27519.903} C_VEL
LIN {X 0,Y 174.265,Z 500.398,A -85,B 0,C 180,E1 -27520.449,E2 -27520.449} C_VEL
LIN {X 0,Y 176.485,Z 484.178,A -85,B 0,C 180,E1 -27520.855,E2 -27520.855} C_VEL
LIN {X 0,Y 176.692,Z 481.646,A -85,B 0,C 180,E1 -27520.985,E2 -27520.985} C_VEL
LIN {X 0,Y 175.292,Z 476.417,A -85,B 0,C 180,E1 -27523.49,E2 -27523.49} C_VEL
LIN {X 0,Y 173.678,Z 472.523,A -85,B 0,C 180,E1 -27526.695,E2 -27526.695} C_VEL
LIN {X 0,Y 172.494,Z 469.612,A -85,B 0,C 180,E1 -27529.947,E2 -27529.947} C_VEL
LIN {X 0,Y 171.587,Z 466.402,A -85,B 0,C 180,E1 -27535.302,E2 -27535.302} C_VEL
LIN {X 0,Y 171.622,Z 466.262,A -85,B 0,C 180,E1 -27539.307,E2 -27539.307} C_VEL
LIN {X 0,Y 172.782,Z 470.178,A -85,B 0,C 180,E1 -27545.362,E2 -27545.362} C_VEL
LIN {X 0,Y 174.186,Z 473.744,A -85,B 0,C 180,E1 -27548.85,E2 -27548.85} C_VEL
LIN {X 0,Y 176.045,Z 478.088,A -85,B 0,C 180,E1 -27552.173,E2 -27552.173} C_VEL
LIN {X 0,Y 176.838,Z 480.156,A -85,B 0,C 180,E1 -27553.401,E2 -27553.401} C_VEL
LIN {X 0,Y 174.64,Z 496.972,A -85,B 0,C 180,E1 -27553.873,E2 -27553.873} C_VEL
LIN {X 0,Y 171.467,Z 511.235,A -85,B 0,C 180,E1 -27554.48,E2 -27554.48} C_VEL
LIN {X 0,Y 167.158,Z 524.944,A -85,B 0,C 180,E1 -27555.344,E2 -27555.344} C_VEL
LIN {X 0,Y 162.013,Z 537.291,A -85,B 0,C 180,E1 -27556.314,E2 -27556.314} C_VEL
LIN {X 0,Y 155.756,Z 549.415,A -85,B 0,C 180,E1 -27557.603,E2 -27557.603} C_VEL
LIN {X 0,Y 148.82,Z 560.542,A -85,B 0,C 180,E1 -27559.184,E2 -27559.184} C_VEL
LIN {X 0,Y 141.239,Z 570.791,A -85,B 0,C 180,E1 -27561.098,E2 -27561.098} C_VEL
LIN {X 0,Y 132.34,Z 580.935,A -85,B 0,C 180,E1 -27563.645,E2 -27563.645} C_VEL
LIN {X 0,Y 123.976,Z 589.226,A -85,B 0,C 180,E1 -27566.611,E2 -27566.611} C_VEL
LIN {X 0,Y 115.778,Z 596.324,A -85,B 0,C 180,E1 -27570.119,E2 -27570.119} C_VEL
LIN {X 0,Y 106.883,Z 602.936,A -85,B 0,C 180,E1 -27574.724,E2 -27574.724} C_VEL
LIN {X 0,Y 97.494,Z 608.858,A -85,B 0,C 180,E1 -27581.014,E2 -27581.014} C_VEL
LIN {X 0,Y 91.573,Z 612.134,A -85,B 0,C 180,E1 -27586.314,E2 -27586.314} C_VEL
LIN {X 0,Y 84.888,Z 615.246,A -85,B 0,C 180,E1 -27594.583,E2 -27594.583} C_VEL
LIN {X 0,Y 80.06,Z 616.967,A -85,B 0,C 180,E1 -27603.966,E2 -27603.966} C_VEL
LIN {X 0,Y 77.252,Z 617.349,A -85,B 0,C 180,E1 -27614.162,E2 -27614.162} C_VEL
LIN {X 0,Y 76.612,Z 616.403,A -85,B 0,C 180,E1 -27624.737,E2 -27624.737} C_VEL
LIN {X 0,Y 76.906,Z 615.438,A -85,B 0,C 180,E1 -27630,E2 -27630} C_VEL
LIN {X 0,Y 78.617,Z 612.507,A -85,B 0,C 180,E1 -27640.299,E2 -27640.299} C_VEL
LIN {X 0,Y 82.263,Z 608.155,A -85,B 0,C 180,E1 -27649.982,E2 -27649.982} C_VEL
LIN {X 0,Y 86.263,Z 603.843,A -85,B 0,C 180,E1 -27656.621,E2 -27656.621} C_VEL
LIN {X 0,Y 92.199,Z 597.581,A -85,B 0,C 180,E1 -27663.547,E2 -27663.547} C_VEL
LIN {X 0,Y 99.077,Z 589.806,A -85,B 0,C 180,E1 -27669.672,E2 -27669.672} C_VEL
LIN {X 0,Y 105.816,Z 581.673,A -85,B 0,C 180,E1 -27674.215,E2 -27674.215} C_VEL
LIN {X 0,Y 113.094,Z 571.878,A -85,B 0,C 180,E1 -27678.218,E2 -27678.218} C_VEL
LIN {X 0,Y 120.101,Z 561.006,A -85,B 0,C 180,E1 -27681.503,E2 -27681.503} C_VEL
LIN {X 0,Y 126.812,Z 548.916,A -85,B 0,C 180,E1 -27684.145,E2 -27684.145} C_VEL
LIN {X 0,Y 132.3,Z 536.966,A -85,B 0,C 180,E1 -27686.099,E2 -27686.099} C_VEL
LIN {X 0,Y 137.282,Z 523.735,A -85,B 0,C 180,E1 -27687.637,E2 -27687.637} C_VEL
LIN {X 0,Y 141.266,Z 509.715,A -85,B 0,C 180,E1 -27688.832,E2 -27688.832} C_VEL
LIN {X 0,Y 144.023,Z 495.636,A -85,B 0,C 180,E1 -27689.683,E2 -27689.683} C_VEL
LIN {X 0,Y 146.335,Z 475.15,A -85,B 0,C 180,E1 -27690.42,E2 -27690.42} C_VEL
LIN {X 0,Y 148.139,Z 456.521,A -85,B 0,C 180,E1 -27691.014,E2 -27691.014} C_VEL
LIN {X 0,Y 145.047,Z 449.263,A -85,B 0,C 180,E1 -27694.6,E2 -27694.6} C_VEL
LIN {X 0,Y 142.214,Z 443.307,A -85,B 0,C 180,E1 -27698.519,E2 -27698.519} C_VEL
LIN {X 0,Y 140.42,Z 439.844,A -85,B 0,C 180,E1 -27701.533,E2 -27701.533} C_VEL
LIN {X 0,Y 139.26,Z 437.666,A -85,B 0,C 180,E1 -27703.882,E2 -27703.882} C_VEL
LIN {X 0,Y 137.694,Z 434.313,A -85,B 0,C 180,E1 -27708.218,E2 -27708.218} C_VEL
LIN {X 0,Y 136.467,Z 431.811,A -85,B 0,C 180,E1 -27716.458,E2 -27716.458} C_VEL
LIN {X 0,Y 136.564,Z 432.074,A -85,B 0,C 180,E1 -27719.362,E2 -27719.362} C_VEL
LIN {X 0,Y 137.837,Z 434.444,A -85,B 0,C 180,E1 -27725.852,E2 -27725.852} C_VEL
LIN {X 0,Y 139.97,Z 438.878,A -85,B 0,C 180,E1 -27731.218,E2 -27731.218} C_VEL
LIN {X 0,Y 142.281,Z 443.381,A -85,B 0,C 180,E1 -27735.212,E2 -27735.212} C_VEL
LIN {X 0,Y 145.029,Z 449.107,A -85,B 0,C 180,E1 -27739,E2 -27739} C_VEL
LIN {X 0,Y 146.761,Z 453.475,A -85,B 0,C 180,E1 -27741.128,E2 -27741.128} C_VEL
LIN {X 0,Y 148.022,Z 457.991,A -85,B 0,C 180,E1 -27742.69,E2 -27742.69} C_VEL
LIN {X 0,Y 144.162,Z 496.293,A -85,B 0,C 180,E1 -27743.948,E2 -27743.948} C_VEL
LIN {X 0,Y 141.525,Z 510.574,A -85,B 0,C 180,E1 -27744.684,E2 -27744.684} C_VEL
LIN {X 0,Y 137.91,Z 523.891,A -85,B 0,C 180,E1 -27745.665,E2 -27745.665} C_VEL
LIN {X 0,Y 133.125,Z 537.175,A -85,B 0,C 180,E1 -27747.021,E2 -27747.021} C_VEL
LIN {X 0,Y 127.347,Z 549.982,A -85,B 0,C 180,E1 -27748.827,E2 -27748.827} C_VEL
LIN {X 0,Y 121.165,Z 561.604,A -85,B 0,C 180,E1 -27751.149,E2 -27751.149} C_VEL
LIN {X 0,Y 114.491,Z 572.342,A -85,B 0,C 180,E1 -27754.038,E2 -27754.038} C_VEL
LIN {X 0,Y 106.832,Z 582.928,A -85,B 0,C 180,E1 -27757.87,E2 -27757.87} C_VEL
LIN {X 0,Y 99.765,Z 591.661,A -85,B 0,C 180,E1 -27762.298,E2 -27762.298} C_VEL
LIN {X 0,Y 92.499,Z 600.034,A -85,B 0,C 180,E1 -27768.333,E2 -27768.333} C_VEL
LIN {X 0,Y 86.368,Z 606.75,A -85,B 0,C 180,E1 -27775.278,E2 -27775.278} C_VEL
LIN {X 0,Y 81.094,Z 612.706,A -85,B 0,C 180,E1 -27784.322,E2 -27784.322} C_VEL
LIN {X 0,Y 77.831,Z 617.06,A -85,B 0,C 180,E1 -27794.283,E2 -27794.283} C_VEL
LIN {X 0,Y 76.656,Z 619.944,A -85,B 0,C 180,E1 -27804.74,E2 -27804.74} C_VEL
LIN {X 0,Y 76.773,Z 620.862,A -85,B 0,C 180,E1 -27810,E2 -27810} C_VEL
LIN {X 0,Y 77.046,Z 621.637,A -85,B 0,C 180,E1 -27820.512,E2 -27820.512} C_VEL
LIN {X 0,Y 79.305,Z 621.088,A -85,B 0,C 180,E1 -27830.761,E2 -27830.761} C_VEL
LIN {X 0,Y 83.832,Z 619.227,A -85,B 0,C 180,E1 -27840.198,E2 -27840.198} C_VEL
LIN {X 0,Y 90.225,Z 616.01,A -85,B 0,C 180,E1 -27848.546,E2 -27848.546} C_VEL
LIN {X 0,Y 98.305,Z 611.319,A -85,B 0,C 180,E1 -27855.635,E2 -27855.635} C_VEL
LIN {X 0,Y 107.702,Z 605.016,A -85,B 0,C 180,E1 -27861.538,E2 -27861.538} C_VEL
LIN {X 0,Y 116.761,Z 598.024,A -85,B 0,C 180,E1 -27865.854,E2 -27865.854} C_VEL
LIN {X 0,Y 126.391,Z 589.381,A -85,B 0,C 180,E1 -27869.526,E2 -27869.526} C_VEL
LIN {X 0,Y 134.972,Z 580.368,A -85,B 0,C 180,E1 -27872.272,E2 -27872.272} C_VEL
LIN {X 0,Y 143.89,Z 569.471,A -85,B 0,C 180,E1 -27874.631,E2 -27874.631} C_VEL
LIN {X 0,Y 151.481,Z 558.423,A -85,B 0,C 180,E1 -27876.388,E2 -27876.388} C_VEL
LIN {X 0,Y 158.491,Z 546.27,A -85,B 0,C 180,E1 -27877.765,E2 -27877.765} C_VEL
LIN {X 0,Y 164.802,Z 532.64,A -85,B 0,C 180,E1 -27878.882,E2 -27878.882} C_VEL
LIN {X 0,Y 166.561,Z 528.22,A -85,B 0,C 180,E1 -27879.164,E2 -27879.164} C_VEL
LIN {X 0,Y 168.295,Z 522.784,A -85,B 0,C 180,E1 -27879.696,E2 -27879.696} C_VEL
LIN {X 0,Y 170.162,Z 513.918,A -85,B 0,C 180,E1 -27881.062,E2 -27881.062} C_VEL
LIN {X 0,Y 171.621,Z 504.882,A -85,B 0,C 180,E1 -27882.33,E2 -27882.33} C_VEL
LIN {X 0,Y 172.554,Z 499.181,A -85,B 0,C 180,E1 -27882.733,E2 -27882.733} C_VEL
LIN {X 0,Y 174.461,Z 485.392,A -85,B 0,C 180,E1 -27883.088,E2 -27883.088} C_VEL
LIN {X 0,Y 173.5,Z 481.857,A -85,B 0,C 180,E1 -27885.066,E2 -27885.066} C_VEL
LIN {X 0,Y 172.277,Z 478.79,A -85,B 0,C 180,E1 -27887.858,E2 -27887.858} C_VEL
LIN {X 0,Y 171.511,Z 476.575,A -85,B 0,C 180,E1 -27890.269,E2 -27890.269} C_VEL
LIN {X 0,Y 170.68,Z 473.376,A -85,B 0,C 180,E1 -27895.869,E2 -27895.869} C_VEL
LIN {X 0,Y 170.73,Z 473.361,A -85,B 0,C 180,E1 -27899.129,E2 -27899.129} C_VEL
LIN {X 0,Y 171.716,Z 477.021,A -85,B 0,C 180,E1 -27904.843,E2 -27904.843} C_VEL
LIN {X 0,Y 173.003,Z 480.604,A -85,B 0,C 180,E1 -27908.322,E2 -27908.322} C_VEL
LIN {X 0,Y 174.523,Z 484.494,A -85,B 0,C 180,E1 -27911.281,E2 -27911.281} C_VEL
LIN {X 0,Y 172.245,Z 499.757,A -85,B 0,C 180,E1 -27911.699,E2 -27911.699} C_VEL
LIN {X 0,Y 168.668,Z 514.245,A -85,B 0,C 180,E1 -27912.339,E2 -27912.339} C_VEL
LIN {X 0,Y 163.795,Z 528.348,A -85,B 0,C 180,E1 -27913.236,E2 -27913.236} C_VEL
LIN {X 0,Y 157.73,Z 541.628,A -85,B 0,C 180,E1 -27914.282,E2 -27914.282} C_VEL
LIN {X 0,Y 150.554,Z 554.269,A -85,B 0,C 180,E1 -27915.684,E2 -27915.684} C_VEL
LIN {X 0,Y 143.055,Z 565.115,A -85,B 0,C 180,E1 -27917.264,E2 -27917.264} C_VEL
LIN {X 0,Y 135.72,Z 574.193,A -85,B 0,C 180,E1 -27919.088,E2 -27919.088} C_VEL
LIN {X 0,Y 126.634,Z 583.8,A -85,B 0,C 180,E1 -27921.631,E2 -27921.631} C_VEL
LIN {X 0,Y 116.487,Z 592.949,A -85,B 0,C 180,E1 -27925.181,E2 -27925.181} C_VEL
LIN {X 0,Y 108.212,Z 599.337,A -85,B 0,C 180,E1 -27928.747,E2 -27928.747} C_VEL
LIN {X 0,Y 100.381,Z 604.577,A -85,B 0,C 180,E1 -27932.846,E2 -27932.846} C_VEL
LIN {X 0,Y 92.632,Z 609.075,A -85,B 0,C 180,E1 -27937.853,E2 -27937.853} C_VEL
LIN {X 0,Y 86.494,Z 612.234,A -85,B 0,C 180,E1 -27943.007,E2 -27943.007} C_VEL
LIN {X 0,Y 79.112,Z 615.389,A -85,B 0,C 180,E1 -27951.55,E2 -27951.55} C_VEL
LIN {X 0,Y 73.646,Z 617.146,A -85,B 0,C 180,E1 -27961.501,E2 -27961.501} C_VEL
LIN {X 0,Y 70.359,Z 617.562,A -85,B 0,C 180,E1 -27972.563,E2 -27972.563} C_VEL
LIN {X 0,Y 69.511,Z 616.649,A -85,B 0,C 180,E1 -27984.197,E2 -27984.197} C_VEL
LIN {X 0,Y 69.782,Z 615.701,A -85,B 0,C 180,E1 -27990,E2 -27990} C_VEL
LIN {X 0,Y 70.488,Z 614.423,A -85,B 0,C 180,E1 -27995.722,E2 -27995.722} C_VEL
LIN {X 0,Y 73.377,Z 610.833,A -85,B 0,C 180,E1 -28006.698,E2 -28006.698} C_VEL
LIN {X 0,Y 78.403,Z 605.76,A -85,B 0,C 180,E1 -28016.627,E2 -28016.627} C_VEL
LIN {X 0,Y 83.558,Z 600.832,A -85,B 0,C 180,E1 -28023.141,E2 -28023.141} C_VEL
LIN {X 0,Y 90.516,Z 593.784,A -85,B 0,C 180,E1 -28029.832,E2 -28029.832} C_VEL
LIN {X 0,Y 97.223,Z 586.419,A -85,B 0,C 180,E1 -28034.812,E2 -28034.812} C_VEL
LIN {X 0,Y 104.624,Z 577.561,A -85,B 0,C 180,E1 -28039.085,E2 -28039.085} C_VEL
LIN {X 0,Y 112.499,Z 566.836,A -85,B 0,C 180,E1 -28042.796,E2 -28042.796} C_VEL
LIN {X 0,Y 119.317,Z 555.976,A -85,B 0,C 180,E1 -28045.548,E2 -28045.548} C_VEL
LIN {X 0,Y 125.608,Z 544.086,A -85,B 0,C 180,E1 -28047.805,E2 -28047.805} C_VEL
LIN {X 0,Y 131.432,Z 530.857,A -85,B 0,C 180,E1 -28049.567,E2 -28049.567} C_VEL
LIN {X 0,Y 135.852,Z 518.088,A -85,B 0,C 180,E1 -28050.805,E2 -28050.805} C_VEL
LIN {X 0,Y 139.518,Z 503.475,A -85,B 0,C 180,E1 -28051.852,E2 -28051.852} C_VEL
LIN {X 0,Y 141.817,Z 489.597,A -85,B 0,C 180,E1 -28052.494,E2 -28052.494} C_VEL
LIN {X 0,Y 144.846,Z 459.916,A -85,B 0,C 180,E1 -28053.448,E2 -28053.448} C_VEL
LIN {X 0,Y 141.964,Z 452.832,A -85,B 0,C 180,E1 -28057.351,E2 -28057.351} C_VEL
LIN {X 0,Y 139.61,Z 447.622,A -85,B 0,C 180,E1 -28061.262,E2 -28061.262} C_VEL
LIN {X 0,Y 138.065,Z 444.503,A -85,B 0,C 180,E1 -28064.498,E2 -28064.498} C_VEL
LIN {X 0,Y 136.556,Z 441.151,A -85,B 0,C 180,E1 -28069.059,E2 -28069.059} C_VEL
LIN {X 0,Y 135.598,Z 438.88,A -85,B 0,C 180,E1 -28076.435,E2 -28076.435} C_VEL
LIN {X 0,Y 135.685,Z 439.209,A -85,B 0,C 180,E1 -28079.357,E2 -28079.357} C_VEL
LIN {X 0,Y 136.715,Z 441.227,A -85,B 0,C 180,E1 -28085.084,E2 -28085.084} C_VEL
LIN {X 0,Y 138.711,Z 445.763,A -85,B 0,C 180,E1 -28090.582,E2 -28090.582} C_VEL
LIN {X 0,Y 141.001,Z 450.548,A -85,B 0,C 180,E1 -28094.776,E2 -28094.776} C_VEL
LIN {X 0,Y 143.437,Z 456.292,A -85,B 0,C 180,E1 -28098.362,E2 -28098.362} C_VEL
LIN {X 0,Y 144.432,Z 459.308,A -85,B 0,C 180,E1 -28099.728,E2 -28099.728} C_VEL
LIN {X 0,Y 144.804,Z 461.279,A -85,B 0,C 180,E1 -28100.319,E2 -28100.319} C_VEL
LIN {X 0,Y 141.001,Z 496.671,A -85,B 0,C 180,E1 -28101.394,E2 -28101.394} C_VEL
LIN {X 0,Y 138.196,Z 511.138,A -85,B 0,C 180,E1 -28102.127,E2 -28102.127} C_VEL
LIN {X 0,Y 134.215,Z 525.043,A -85,B 0,C 180,E1 -28103.131,E2 -28103.131} C_VEL
LIN {X 0,Y 129.294,Z 538.032,A -85,B 0,C 180,E1 -28104.433,E2 -28104.433} C_VEL
LIN {X 0,Y 123.33,Z 550.635,A -85,B 0,C 180,E1 -28106.169,E2 -28106.169} C_VEL
LIN {X 0,Y 116.88,Z 562.158,A -85,B 0,C 180,E1 -28108.435,E2 -28108.435} C_VEL
LIN {X 0,Y 110.646,Z 571.741,A -85,B 0,C 180,E1 -28110.967,E2 -28110.967} C_VEL
LIN {X 0,Y 103.92,Z 580.752,A -85,B 0,C 180,E1 -28114.063,E2 -28114.063} C_VEL
LIN {X 0,Y 96.272,Z 589.81,A -85,B 0,C 180,E1 -28118.303,E2 -28118.303} C_VEL
LIN {X 0,Y 88.346,Z 598.49,A -85,B 0,C 180,E1 -28124.28,E2 -28124.28} C_VEL
LIN {X 0,Y 82.225,Z 604.649,A -85,B 0,C 180,E1 -28130.285,E2 -28130.285} C_VEL
LIN {X 0,Y 75.993,Z 611.034,A -85,B 0,C 180,E1 -28139.427,E2 -28139.427} C_VEL
LIN {X 0,Y 71.658,Z 615.838,A -85,B 0,C 180,E1 -28149.925,E2 -28149.925} C_VEL
LIN {X 0,Y 69.998,Z 618.404,A -85,B 0,C 180,E1 -28158.416,E2 -28158.416} C_VEL
LIN {X 0,Y 69.668,Z 620.619,A -85,B 0,C 180,E1 -28170,E2 -28170} C_VEL
LIN {X 0,Y 70.047,Z 621.426,A -85,B 0,C 180,E1 -28181.576,E2 -28181.576} C_VEL
LIN {X 0,Y 72.659,Z 620.909,A -85,B 0,C 180,E1 -28192.761,E2 -28192.761} C_VEL
LIN {X 0,Y 77.738,Z 619.081,A -85,B 0,C 180,E1 -28202.849,E2 -28202.849} C_VEL
LIN {X 0,Y 85.427,Z 615.562,A -85,B 0,C 180,E1 -28212.235,E2 -28212.235} C_VEL
LIN {X 0,Y 93.446,Z 611.261,A -85,B 0,C 180,E1 -28218.77,E2 -28218.77} C_VEL
LIN {X 0,Y 103.409,Z 604.998,A -85,B 0,C 180,E1 -28224.641,E2 -28224.641} C_VEL
LIN {X 0,Y 112.914,Z 598.048,A -85,B 0,C 180,E1 -28228.849,E2 -28228.849} C_VEL
LIN {X 0,Y 122.942,Z 589.454,A -85,B 0,C 180,E1 -28232.379,E2 -28232.379} C_VEL
LIN {X 0,Y 131.817,Z 580.496,A -85,B 0,C 180,E1 -28235.006,E2 -28235.006} C_VEL
LIN {X 0,Y 139.443,Z 571.614,A -85,B 0,C 180,E1 -28236.894,E2 -28236.894} C_VEL
LIN {X 0,Y 147.992,Z 559.872,A -85,B 0,C 180,E1 -28238.74,E2 -28238.74} C_VEL
LIN {X 0,Y 155.166,Z 548.102,A -85,B 0,C 180,E1 -28240.02,E2 -28240.02} C_VEL
LIN {X 0,Y 161.582,Z 535.129,A -85,B 0,C 180,E1 -28241.083,E2 -28241.083} C_VEL
LIN {X 0,Y 166.82,Z 521.608,A -85,B 0,C 180,E1 -28241.882,E2 -28241.882} C_VEL
LIN {X 0,Y 170.883,Z 507.233,A -85,B 0,C 180,E1 -28242.494,E2 -28242.494} C_VEL
LIN {X 0,Y 172.554,Z 499.181,A -85,B 0,C 180,E1 -28242.733,E2 -28242.733} C_VEL
LIN {X 0,Y 172.923,Z 496.06,A -85,B 0,C 180,E1 -28243.059,E2 -28243.059} C_VEL
LIN {X 0,Y 172.873,Z 492.829,A -85,B 0,C 180,E1 -28243.854,E2 -28243.854} C_VEL
LIN {X 0,Y 172.446,Z 489.848,A -85,B 0,C 180,E1 -28245.121,E2 -28245.121} C_VEL
LIN {X 0,Y 171.573,Z 486.707,A -85,B 0,C 180,E1 -28247.308,E2 -28247.308} C_VEL
LIN {X 0,Y 171.226,Z 485.771,A -85,B 0,C 180,E1 -28248.233,E2 -28248.233} C_VEL
LIN {X 0,Y 170.461,Z 483.443,A -85,B 0,C 180,E1 -28250.838,E2 -28250.838} C_VEL
LIN {X 0,Y 169.79,Z 480.345,A -85,B 0,C 180,E1 -28256.441,E2 -28256.441} C_VEL
LIN {X 0,Y 169.839,Z 480.338,A -85,B 0,C 180,E1 -28258.774,E2 -28258.774} C_VEL
LIN {X 0,Y 170.635,Z 483.796,A -85,B 0,C 180,E1 -28264.217,E2 -28264.217} C_VEL
LIN {X 0,Y 171.877,Z 487.629,A -85,B 0,C 180,E1 -28267.934,E2 -28267.934} C_VEL
LIN {X 0,Y 172.372,Z 489.08,A -85,B 0,C 180,E1 -28269.119,E2 -28269.119} C_VEL
LIN {X 0,Y 169.761,Z 503.622,A -85,B 0,C 180,E1 -28269.515,E2 -28269.515} C_VEL
LIN {X 0,Y 165.813,Z 518.016,A -85,B 0,C 180,E1 -28270.175,E2 -28270.175} C_VEL
LIN {X 0,Y 161.062,Z 530.704,A -85,B 0,C 180,E1 -28270.958,E2 -28270.958} C_VEL
LIN {X 0,Y 155.296,Z 542.746,A -85,B 0,C 180,E1 -28271.869,E2 -28271.869} C_VEL
LIN {X 0,Y 147.966,Z 555.212,A -85,B 0,C 180,E1 -28273.177,E2 -28273.177} C_VEL
LIN {X 0,Y 139.365,Z 567.087,A -85,B 0,C 180,E1 -28274.855,E2 -28274.855} C_VEL
LIN {X 0,Y 130.378,Z 577.446,A -85,B 0,C 180,E1 -28276.906,E2 -28276.906} C_VEL
LIN {X 0,Y 121.102,Z 586.509,A -85,B 0,C 180,E1 -28279.435,E2 -28279.435} C_VEL
LIN {X 0,Y 110.674,Z 595.151,A -85,B 0,C 180,E1 -28282.964,E2 -28282.964} C_VEL
LIN {X 0,Y 102.122,Z 601.187,A -85,B 0,C 180,E1 -28286.539,E2 -28286.539} C_VEL
LIN {X 0,Y 91.388,Z 607.586,A -85,B 0,C 180,E1 -28292.231,E2 -28292.231} C_VEL
LIN {X 0,Y 81.738,Z 612.326,A -85,B 0,C 180,E1 -28299.302,E2 -28299.302} C_VEL
LIN {X 0,Y 73.597,Z 615.532,A -85,B 0,C 180,E1 -28308.054,E2 -28308.054} C_VEL
LIN {X 0,Y 67.402,Z 617.324,A -85,B 0,C 180,E1 -28318.578,E2 -28318.578} C_VEL
LIN {X 0,Y 63.535,Z 617.775,A -85,B 0,C 180,E1 -28330.619,E2 -28330.619} C_VEL
LIN {X 0,Y 62.411,Z 616.896,A -85,B 0,C 180,E1 -28343.534,E2 -28343.534} C_VEL
LIN {X 0,Y 62.681,Z 615.964,A -85,B 0,C 180,E1 -28350,E2 -28350} C_VEL
LIN {X 0,Y 63.444,Z 614.702,A -85,B 0,C 180,E1 -28356.36,E2 -28356.36} C_VEL
LIN {X 0,Y 66.641,Z 611.148,A -85,B 0,C 180,E1 -28368.444,E2 -28368.444} C_VEL
LIN {X 0,Y 72.144,Z 606.114,A -85,B 0,C 180,E1 -28379.148,E2 -28379.148} C_VEL
LIN {X 0,Y 77.741,Z 601.227,A -85,B 0,C 180,E1 -28385.987,E2 -28385.987} C_VEL
LIN {X 0,Y 85.207,Z 594.226,A -85,B 0,C 180,E1 -28392.879,E2 -28392.879} C_VEL
LIN {X 0,Y 92.334,Z 586.912,A -85,B 0,C 180,E1 -28397.91,E2 -28397.91} C_VEL
LIN {X 0,Y 100.147,Z 578.112,A -85,B 0,C 180,E1 -28402.135,E2 -28402.135} C_VEL
LIN {X 0,Y 108.377,Z 567.457,A -85,B 0,C 180,E1 -28405.77,E2 -28405.77} C_VEL
LIN {X 0,Y 115.464,Z 556.684,A -85,B 0,C 180,E1 -28408.443,E2 -28408.443} C_VEL
LIN {X 0,Y 121.992,Z 544.902,A -85,B 0,C 180,E1 -28410.613,E2 -28410.613} C_VEL
LIN {X 0,Y 128.009,Z 531.867,A -85,B 0,C 180,E1 -28412.285,E2 -28412.285} C_VEL
LIN {X 0,Y 132.936,Z 518.116,A -85,B 0,C 180,E1 -28413.562,E2 -28413.562} C_VEL
LIN {X 0,Y 136.461,Z 504.608,A -85,B 0,C 180,E1 -28414.506,E2 -28414.506} C_VEL
LIN {X 0,Y 138.907,Z 490.768,A -85,B 0,C 180,E1 -28415.129,E2 -28415.129} C_VEL
LIN {X 0,Y 141.83,Z 463.465,A -85,B 0,C 180,E1 -28415.962,E2 -28415.962} C_VEL
LIN {X 0,Y 139.58,Z 457.681,A -85,B 0,C 180,E1 -28419.505,E2 -28419.505} C_VEL
LIN {X 0,Y 137.832,Z 453.508,A -85,B 0,C 180,E1 -28422.883,E2 -28422.883} C_VEL
LIN {X 0,Y 136.671,Z 450.996,A -85,B 0,C 180,E1 -28425.664,E2 -28425.664} C_VEL
LIN {X 0,Y 135.508,Z 448.031,A -85,B 0,C 180,E1 -28429.691,E2 -28429.691} C_VEL
LIN {X 0,Y 134.739,Z 445.846,A -85,B 0,C 180,E1 -28437.009,E2 -28437.009} C_VEL
LIN {X 0,Y 134.824,Z 446.486,A -85,B 0,C 180,E1 -28439.676,E2 -28439.676} C_VEL
LIN {X 0,Y 135.647,Z 448.162,A -85,B 0,C 180,E1 -28444.46,E2 -28444.46} C_VEL
LIN {X 0,Y 137.297,Z 452.244,A -85,B 0,C 180,E1 -28449.529,E2 -28449.529} C_VEL
LIN {X 0,Y 139.384,Z 457.059,A -85,B 0,C 180,E1 -28453.763,E2 -28453.763} C_VEL
LIN {X 0,Y 141.425,Z 462.28,A -85,B 0,C 180,E1 -28457.067,E2 -28457.067} C_VEL
LIN {X 0,Y 141.843,Z 463.697,A -85,B 0,C 180,E1 -28457.719,E2 -28457.719} C_VEL
LIN {X 0,Y 138.437,Z 495.242,A -85,B 0,C 180,E1 -28458.675,E2 -28458.675} C_VEL
LIN {X 0,Y 135.568,Z 510.044,A -85,B 0,C 180,E1 -28459.343,E2 -28459.343} C_VEL
LIN {X 0,Y 131.572,Z 523.918,A -85,B 0,C 180,E1 -28460.268,E2 -28460.268} C_VEL
LIN {X 0,Y 126.504,Z 537.108,A -85,B 0,C 180,E1 -28461.482,E2 -28461.482} C_VEL
LIN {X 0,Y 120.345,Z 549.85,A -85,B 0,C 180,E1 -28463.11,E2 -28463.11} C_VEL
LIN {X 0,Y 113.637,Z 561.469,A -85,B 0,C 180,E1 -28465.248,E2 -28465.248} C_VEL
LIN {X 0,Y 106.865,Z 571.523,A -85,B 0,C 180,E1 -28467.797,E2 -28467.797} C_VEL
LIN {X 0,Y 98.716,Z 581.86,A -85,B 0,C 180,E1 -28471.317,E2 -28471.317} C_VEL
LIN {X 0,Y 90.73,Z 590.699,A -85,B 0,C 180,E1 -28475.579,E2 -28475.579} C_VEL
LIN {X 0,Y 83.496,Z 598.058,A -85,B 0,C 180,E1 -28480.754,E2 -28480.754} C_VEL
LIN {X 0,Y 76.275,Z 604.779,A -85,B 0,C 180,E1 -28487.485,E2 -28487.485} C_VEL
LIN {X 0,Y 69.923,Z 610.685,A -85,B 0,C 180,E1 -28496.441,E2 -28496.441} C_VEL
LIN {X 0,Y 64.999,Z 615.527,A -85,B 0,C 180,E1 -28507.764,E2 -28507.764} C_VEL
LIN {X 0,Y 63.041,Z 618.128,A -85,B 0,C 180,E1 -28517.117,E2 -28517.117} C_VEL
LIN {X 0,Y 62.558,Z 620.377,A -85,B 0,C 180,E1 -28530,E2 -28530} C_VEL
LIN {X 0,Y 63.091,Z 621.216,A -85,B 0,C 180,E1 -28542.873,E2 -28542.873} C_VEL
LIN {X 0,Y 66.122,Z 620.73,A -85,B 0,C 180,E1 -28555.16,E2 -28555.16} C_VEL
LIN {X 0,Y 71.827,Z 618.935,A -85,B 0,C 180,E1 -28565.949,E2 -28565.949} C_VEL
LIN {X 0,Y 79.762,Z 615.697,A -85,B 0,C 180,E1 -28575.181,E2 -28575.181} C_VEL
LIN {X 0,Y 88.91,Z 611.198,A -85,B 0,C 180,E1 -28582.226,E2 -28582.226} C_VEL
LIN {X 0,Y 99.446,Z 604.979,A -85,B 0,C 180,E1 -28587.999,E2 -28587.999} C_VEL
LIN {X 0,Y 109.405,Z 598.074,A -85,B 0,C 180,E1 -28592.038,E2 -28592.038} C_VEL
LIN {X 0,Y 119.817,Z 589.531,A -85,B 0,C 180,E1 -28595.388,E2 -28595.388} C_VEL
LIN {X 0,Y 128.975,Z 580.631,A -85,B 0,C 180,E1 -28597.869,E2 -28597.869} C_VEL
LIN {X 0,Y 136.822,Z 571.815,A -85,B 0,C 180,E1 -28599.62,E2 -28599.62} C_VEL
LIN {X 0,Y 145.575,Z 560.155,A -85,B 0,C 180,E1 -28601.338,E2 -28601.338} C_VEL
LIN {X 0,Y 152.889,Z 548.49,A -85,B 0,C 180,E1 -28602.517,E2 -28602.517} C_VEL
LIN {X 0,Y 159.43,Z 535.658,A -85,B 0,C 180,E1 -28603.488,E2 -28603.488} C_VEL
LIN {X 0,Y 165.03,Z 521.613,A -85,B 0,C 180,E1 -28604.254,E2 -28604.254} C_VEL
LIN {X 0,Y 169.191,Z 507.226,A -85,B 0,C 180,E1 -28604.818,E2 -28604.818} C_VEL
LIN {X 0,Y 171.87,Z 493.43,A -85,B 0,C 180,E1 -28605.163,E2 -28605.163} C_VEL
LIN {X 0,Y 172.391,Z 489.328,A -85,B 0,C 180,E1 -28605.306,E2 -28605.306} C_VEL
LIN {X 0,Y 171.931,Z 487.797,A -85,B 0,C 180,E1 -28606.407,E2 -28606.407} C_VEL
LIN {X 0,Y 171.226,Z 485.771,A -85,B 0,C 180,E1 -28608.233,E2 -28608.233} C_VEL
LIN {X 0,Y 170.706,Z 485.346,A -85,B 0,C 180,E1 -28609.539,E2 -28609.539} C_VEL
LIN {X 0,Y 169.786,Z 486.645,A -85,B 0,C 180,E1 -28611.737,E2 -28611.737} C_VEL
LIN {X 0,Y 169.088,Z 488.152,A -85,B 0,C 180,E1 -28613.971,E2 -28613.971} C_VEL
LIN {X 0,Y 168.92,Z 488.024,A -85,B 0,C 180,E1 -28615.331,E2 -28615.331} C_VEL
LIN {X 0,Y 168.919,Z 487.328,A -85,B 0,C 180,E1 -28616.873,E2 -28616.873} C_VEL
LIN {X 0,Y 168.947,Z 487.675,A -85,B 0,C 180,E1 -28618.943,E2 -28618.943} C_VEL
LIN {X 0,Y 169.527,Z 490.686,A -85,B 0,C 180,E1 -28623.733,E2 -28623.733} C_VEL
LIN {X 0,Y 170.346,Z 493.827,A -85,B 0,C 180,E1 -28626.843,E2 -28626.843} C_VEL
LIN {X 0,Y 167.345,Z 508.053,A -85,B 0,C 180,E1 -28627.323,E2 -28627.323} C_VEL
LIN {X 0,Y 163.208,Z 521.496,A -85,B 0,C 180,E1 -28627.951,E2 -28627.951} C_VEL
LIN {X 0,Y 158.171,Z 533.842,A -85,B 0,C 180,E1 -28628.658,E2 -28628.658} C_VEL
LIN {X 0,Y 151.494,Z 546.769,A -85,B 0,C 180,E1 -28629.672,E2 -28629.672} C_VEL
LIN {X 0,Y 144.004,Z 558.471,A -85,B 0,C 180,E1 -28630.84,E2 -28630.84} C_VEL
LIN {X 0,Y 136.599,Z 568.189,A -85,B 0,C 180,E1 -28632.172,E2 -28632.172} C_VEL
LIN {X 0,Y 128.47,Z 577.3,A -85,B 0,C 180,E1 -28633.834,E2 -28633.834} C_VEL
LIN {X 0,Y 118.895,Z 586.421,A -85,B 0,C 180,E1 -28636.152,E2 -28636.152} C_VEL
LIN {X 0,Y 108.062,Z 595.115,A -85,B 0,C 180,E1 -28639.437,E2 -28639.437} C_VEL
LIN {X 0,Y 99.101,Z 601.197,A -85,B 0,C 180,E1 -28642.794,E2 -28642.794} C_VEL
LIN {X 0,Y 87.756,Z 607.637,A -85,B 0,C 180,E1 -28648.247,E2 -28648.247} C_VEL
LIN {X 0,Y 77.367,Z 612.416,A -85,B 0,C 180,E1 -28655.161,E2 -28655.161} C_VEL
LIN {X 0,Y 68.398,Z 615.672,A -85,B 0,C 180,E1 -28664.008,E2 -28664.008} C_VEL
LIN {X 0,Y 61.371,Z 617.502,A -85,B 0,C 180,E1 -28675.07,E2 -28675.07} C_VEL
LIN {X 0,Y 56.8,Z 617.988,A -85,B 0,C 180,E1 -28688.211,E2 -28688.211} C_VEL
LIN {X 0,Y 55.315,Z 617.142,A -85,B 0,C 180,E1 -28702.701,E2 -28702.701} C_VEL
LIN {X 0,Y 55.574,Z 616.227,A -85,B 0,C 180,E1 -28710,E2 -28710} C_VEL
LIN {X 0,Y 56.412,Z 614.982,A -85,B 0,C 180,E1 -28717.156,E2 -28717.156} C_VEL
LIN {X 0,Y 59.971,Z 611.464,A -85,B 0,C 180,E1 -28730.583,E2 -28730.583} C_VEL
LIN {X 0,Y 66.042,Z 606.47,A -85,B 0,C 180,E1 -28742.145,E2 -28742.145} C_VEL
LIN {X 0,Y 72.125,Z 601.624,A -85,B 0,C 180,E1 -28749.298,E2 -28749.298} C_VEL
LIN {X 0,Y 80.176,Z 594.666,A -85,B 0,C 180,E1 -28756.315,E2 -28756.315} C_VEL
LIN {X 0,Y 87.75,Z 587.404,A -85,B 0,C 180,E1 -28761.34,E2 -28761.34} C_VEL
LIN {X 0,Y 95.965,Z 578.661,A -85,B 0,C 180,E1 -28765.474,E2 -28765.474} C_VEL
LIN {X 0,Y 104.572,Z 568.073,A -85,B 0,C 180,E1 -28768.967,E2 -28768.967} C_VEL
LIN {X 0,Y 111.926,Z 557.385,A -85,B 0,C 180,E1 -28771.528,E2 -28771.528} C_VEL
LIN {X 0,Y 118.69,Z 545.707,A -85,B 0,C 180,E1 -28773.582,E2 -28773.582} C_VEL
LIN {X 0,Y 124.886,Z 532.814,A -85,B 0,C 180,E1 -28775.15,E2 -28775.15} C_VEL
LIN {X 0,Y 129.96,Z 519.37,A -85,B 0,C 180,E1 -28776.337,E2 -28776.337} C_VEL
LIN {X 0,Y 133.723,Z 505.741,A -85,B 0,C 180,E1 -28777.251,E2 -28777.251} C_VEL
LIN {X 0,Y 136.367,Z 491.495,A -85,B 0,C 180,E1 -28777.869,E2 -28777.869} C_VEL
LIN {X 0,Y 139.057,Z 467.181,A -85,B 0,C 180,E1 -28778.599,E2 -28778.599} C_VEL
LIN {X 0,Y 137.222,Z 462.072,A -85,B 0,C 180,E1 -28782.102,E2 -28782.102} C_VEL
LIN {X 0,Y 135.588,Z 457.948,A -85,B 0,C 180,E1 -28786.128,E2 -28786.128} C_VEL
LIN {X 0,Y 134.417,Z 454.843,A -85,B 0,C 180,E1 -28790.595,E2 -28790.595} C_VEL
LIN {X 0,Y 133.871,Z 452.906,A -85,B 0,C 180,E1 -28796.99,E2 -28796.99} C_VEL
LIN {X 0,Y 134.074,Z 454.019,A -85,B 0,C 180,E1 -28800.938,E2 -28800.938} C_VEL
LIN {X 0,Y 134.629,Z 455.218,A -85,B 0,C 180,E1 -28803.992,E2 -28803.992} C_VEL
LIN {X 0,Y 135.986,Z 458.909,A -85,B 0,C 180,E1 -28808.614,E2 -28808.614} C_VEL
LIN {X 0,Y 137.646,Z 463.126,A -85,B 0,C 180,E1 -28812.397,E2 -28812.397} C_VEL
LIN {X 0,Y 139.096,Z 467.172,A -85,B 0,C 180,E1 -28815.084,E2 -28815.084} C_VEL
LIN {X 0,Y 135.895,Z 495.647,A -85,B 0,C 180,E1 -28815.918,E2 -28815.918} C_VEL
LIN {X 0,Y 132.896,Z 510.379,A -85,B 0,C 180,E1 -28816.538,E2 -28816.538} C_VEL
LIN {X 0,Y 128.874,Z 523.916,A -85,B 0,C 180,E1 -28817.385,E2 -28817.385} C_VEL
LIN {X 0,Y 124.061,Z 536.172,A -85,B 0,C 180,E1 -28818.405,E2 -28818.405} C_VEL
LIN {X 0,Y 117.74,Z 549.062,A -85,B 0,C 180,E1 -28819.931,E2 -28819.931} C_VEL
LIN {X 0,Y 110.751,Z 560.775,A -85,B 0,C 180,E1 -28821.869,E2 -28821.869} C_VEL
LIN {X 0,Y 103.351,Z 571.411,A -85,B 0,C 180,E1 -28824.434,E2 -28824.434} C_VEL
LIN {X 0,Y 95.201,Z 581.325,A -85,B 0,C 180,E1 -28827.644,E2 -28827.644} C_VEL
LIN {X 0,Y 86.751,Z 590.218,A -85,B 0,C 180,E1 -28831.722,E2 -28831.722} C_VEL
LIN {X 0,Y 78.986,Z 597.625,A -85,B 0,C 180,E1 -28836.796,E2 -28836.796} C_VEL
LIN {X 0,Y 70.569,Z 604.885,A -85,B 0,C 180,E1 -28844.195,E2 -28844.195} C_VEL
LIN {X 0,Y 64.068,Z 610.336,A -85,B 0,C 180,E1 -28852.893,E2 -28852.893} C_VEL
LIN {X 0,Y 58.433,Z 615.216,A -85,B 0,C 180,E1 -28865.106,E2 -28865.106} C_VEL
LIN {X 0,Y 56.099,Z 617.851,A -85,B 0,C 180,E1 -28875.49,E2 -28875.49} C_VEL
LIN {X 0,Y 55.443,Z 619.168,A -85,B 0,C 180,E1 -28882.718,E2 -28882.718} C_VEL
LIN {X 0,Y 55.468,Z 620.135,A -85,B 0,C 180,E1 -28890,E2 -28890} C_VEL
LIN {X 0,Y 56.154,Z 621.005,A -85,B 0,C 180,E1 -28904.496,E2 -28904.496} C_VEL
LIN {X 0,Y 59.729,Z 620.552,A -85,B 0,C 180,E1 -28918.076,E2 -28918.076} C_VEL
LIN {X 0,Y 66.166,Z 618.79,A -85,B 0,C 180,E1 -28929.59,E2 -28929.59} C_VEL
LIN {X 0,Y 74.655,Z 615.677,A -85,B 0,C 180,E1 -28938.86,E2 -28938.86} C_VEL
LIN {X 0,Y 84.72,Z 611.131,A -85,B 0,C 180,E1 -28946.051,E2 -28946.051} C_VEL
LIN {X 0,Y 95.854,Z 604.965,A -85,B 0,C 180,E1 -28951.62,E2 -28951.62} C_VEL
LIN {X 0,Y 106.26,Z 598.104,A -85,B 0,C 180,E1 -28955.422,E2 -28955.422} C_VEL
LIN {X 0,Y 117.041,Z 589.609,A -85,B 0,C 180,E1 -28958.546,E2 -28958.546} C_VEL
LIN {X 0,Y 126.468,Z 580.766,A -85,B 0,C 180,E1 -28960.854,E2 -28960.854} C_VEL
LIN {X 0,Y 134.516,Z 572.017,A -85,B 0,C 180,E1 -28962.454,E2 -28962.454} C_VEL
LIN {X 0,Y 143.467,Z 560.438,A -85,B 0,C 180,E1 -28964.017,E2 -28964.017} C_VEL
LIN {X 0,Y 150.913,Z 548.878,A -85,B 0,C 180,E1 -28965.083,E2 -28965.083} C_VEL
LIN {X 0,Y 157.566,Z 536.186,A -85,B 0,C 180,E1 -28965.954,E2 -28965.954} C_VEL
LIN {X 0,Y 162.753,Z 523.714,A -85,B 0,C 180,E1 -28966.575,E2 -28966.575} C_VEL
LIN {X 0,Y 167.21,Z 509.5,A -85,B 0,C 180,E1 -28967.101,E2 -28967.101} C_VEL
LIN {X 0,Y 170.279,Z 495.104,A -85,B 0,C 180,E1 -28967.458,E2 -28967.458} C_VEL
LIN {X 0,Y 170.434,Z 493.962,A -85,B 0,C 180,E1 -28967.506,E2 -28967.506} C_VEL
LIN {X 0,Y 169.47,Z 490.451,A -85,B 0,C 180,E1 -28971.054,E2 -28971.054} C_VEL
LIN {X 0,Y 168.92,Z 488.024,A -85,B 0,C 180,E1 -28975.331,E2 -28975.331} C_VEL
LIN {X 0,Y 168.832,Z 488.105,A -85,B 0,C 180,E1 -28976.418,E2 -28976.418} C_VEL
LIN {X 0,Y 168.572,Z 489.859,A -85,B 0,C 180,E1 -28977.865,E2 -28977.865} C_VEL
LIN {X 0,Y 168.019,Z 495.173,A -85,B 0,C 180,E1 -28980.631,E2 -28980.631} C_VEL
LIN {X 0,Y 168.009,Z 496.589,A -85,B 0,C 180,E1 -28981.96,E2 -28981.96} C_VEL
LIN {X 0,Y 168.39,Z 498.786,A -85,B 0,C 180,E1 -28984.583,E2 -28984.583} C_VEL
LIN {X 0,Y 164.953,Z 512.822,A -85,B 0,C 180,E1 -28985.084,E2 -28985.084} C_VEL
LIN {X 0,Y 160.242,Z 526.391,A -85,B 0,C 180,E1 -28985.725,E2 -28985.725} C_VEL
LIN {X 0,Y 153.847,Z 540.202,A -85,B 0,C 180,E1 -28986.511,E2 -28986.511} C_VEL
LIN {X 0,Y 147.061,Z 551.916,A -85,B 0,C 180,E1 -28987.428,E2 -28987.428} C_VEL
LIN {X 0,Y 138.774,Z 563.64,A -85,B 0,C 180,E1 -28988.663,E2 -28988.663} C_VEL
LIN {X 0,Y 131.94,Z 571.863,A -85,B 0,C 180,E1 -28989.801,E2 -28989.801} C_VEL
LIN {X 0,Y 121.988,Z 581.959,A -85,B 0,C 180,E1 -28991.656,E2 -28991.656} C_VEL
LIN {X 0,Y 112.247,Z 590.321,A -85,B 0,C 180,E1 -28993.962,E2 -28993.962} C_VEL
LIN {X 0,Y 101.179,Z 598.287,A -85,B 0,C 180,E1 -28997.242,E2 -28997.242} C_VEL
LIN {X 0,Y 90.474,Z 604.667,A -85,B 0,C 180,E1 -29001.231,E2 -29001.231} C_VEL
LIN {X 0,Y 78.861,Z 610.295,A -85,B 0,C 180,E1 -29006.98,E2 -29006.98} C_VEL
LIN {X 0,Y 68.305,Z 614.339,A -85,B 0,C 180,E1 -29014.602,E2 -29014.602} C_VEL
LIN {X 0,Y 59.33,Z 616.916,A -85,B 0,C 180,E1 -29024.706,E2 -29024.706} C_VEL
LIN {X 0,Y 52.536,Z 618.107,A -85,B 0,C 180,E1 -29037.65,E2 -29037.65} C_VEL
LIN {X 0,Y 48.783,Z 617.96,A -85,B 0,C 180,E1 -29053.254,E2 -29053.254} C_VEL
LIN {X 0,Y 48.223,Z 617.388,A -85,B 0,C 180,E1 -29061.62,E2 -29061.62} C_VEL
LIN {X 0,Y 48.458,Z 616.489,A -85,B 0,C 180,E1 -29070,E2 -29070} C_VEL
LIN {X 0,Y 49.381,Z 615.26,A -85,B 0,C 180,E1 -29078.182,E2 -29078.182} C_VEL
LIN {X 0,Y 53.395,Z 611.778,A -85,B 0,C 180,E1 -29093.257,E2 -29093.257} C_VEL
LIN {X 0,Y 60.178,Z 606.821,A -85,B 0,C 180,E1 -29105.726,E2 -29105.726} C_VEL
LIN {X 0,Y 66.808,Z 602.016,A -85,B 0,C 180,E1 -29113.138,E2 -29113.138} C_VEL
LIN {X 0,Y 75.455,Z 595.104,A -85,B 0,C 180,E1 -29120.21,E2 -29120.21} C_VEL
LIN {X 0,Y 84.944,Z 586.543,A -85,B 0,C 180,E1 -29125.827,E2 -29125.827} C_VEL
LIN {X 0,Y 93.61,Z 577.59,A -85,B 0,C 180,E1 -29129.696,E2 -29129.696} C_VEL
LIN {X 0,Y 102.617,Z 566.75,A -85,B 0,C 180,E1 -29132.913,E2 -29132.913} C_VEL
LIN {X 0,Y 110.297,Z 555.746,A -85,B 0,C 180,E1 -29135.226,E2 -29135.226} C_VEL
LIN {X 0,Y 117.294,Z 543.645,A -85,B 0,C 180,E1 -29137.103,E2 -29137.103} C_VEL
LIN {X 0,Y 123.681,Z 530.045,A -85,B 0,C 180,E1 -29138.507,E2 -29138.507} C_VEL
LIN {X 0,Y 128.555,Z 516.597,A -85,B 0,C 180,E1 -29139.526,E2 -29139.526} C_VEL
LIN {X 0,Y 132.136,Z 503.038,A -85,B 0,C 180,E1 -29140.294,E2 -29140.294} C_VEL
LIN {X 0,Y 134.674,Z 488.266,A -85,B 0,C 180,E1 -29140.82,E2 -29140.82} C_VEL
LIN {X 0,Y 136.574,Z 471.028,A -85,B 0,C 180,E1 -29141.334,E2 -29141.334} C_VEL
LIN {X 0,Y 135.005,Z 466.399,A -85,B 0,C 180,E1 -29145.105,E2 -29145.105} C_VEL
LIN {X 0,Y 134.167,Z 464.147,A -85,B 0,C 180,E1 -29147.71,E2 -29147.71} C_VEL
LIN {X 0,Y 133.473,Z 461.841,A -85,B 0,C 180,E1 -29150.91,E2 -29150.91} C_VEL
LIN {X 0,Y 133.002,Z 459.97,A -85,B 0,C 180,E1 -29156.97,E2 -29156.97} C_VEL
LIN {X 0,Y 133.542,Z 461.851,A -85,B 0,C 180,E1 -29163.016,E2 -29163.016} C_VEL
LIN {X 0,Y 134.697,Z 465.514,A -85,B 0,C 180,E1 -29167.635,E2 -29167.635} C_VEL
LIN {X 0,Y 136.102,Z 469.543,A -85,B 0,C 180,E1 -29171.259,E2 -29171.259} C_VEL
LIN {X 0,Y 136.616,Z 471.03,A -85,B 0,C 180,E1 -29172.364,E2 -29172.364} C_VEL
LIN {X 0,Y 133.665,Z 496.014,A -85,B 0,C 180,E1 -29173.053,E2 -29173.053} C_VEL
LIN {X 0,Y 130.556,Z 510.714,A -85,B 0,C 180,E1 -29173.629,E2 -29173.629} C_VEL
LIN {X 0,Y 126.108,Z 525.05,A -85,B 0,C 180,E1 -29174.469,E2 -29174.469} C_VEL
LIN {X 0,Y 120.37,Z 538.792,A -85,B 0,C 180,E1 -29175.56,E2 -29175.56} C_VEL
LIN {X 0,Y 113.879,Z 551.136,A -85,B 0,C 180,E1 -29176.953,E2 -29176.953} C_VEL
LIN {X 0,Y 106.726,Z 562.456,A -85,B 0,C 180,E1 -29178.813,E2 -29178.813} C_VEL
LIN {X 0,Y 98.202,Z 573.827,A -85,B 0,C 180,E1 -29181.513,E2 -29181.513} C_VEL
LIN {X 0,Y 89.089,Z 583.966,A -85,B 0,C 180,E1 -29184.882,E2 -29184.882} C_VEL
LIN {X 0,Y 80.383,Z 592.385,A -85,B 0,C 180,E1 -29189.039,E2 -29189.039} C_VEL
LIN {X 0,Y 71.002,Z 600.436,A -85,B 0,C 180,E1 -29195.255,E2 -29195.255} C_VEL
LIN {X 0,Y 62.626,Z 606.909,A -85,B 0,C 180,E1 -29203.162,E2 -29203.162} C_VEL
LIN {X 0,Y 54.943,Z 612.643,A -85,B 0,C 180,E1 -29214.859,E2 -29214.859} C_VEL
LIN {X 0,Y 50.903,Z 615.884,A -85,B 0,C 180,E1 -29225.532,E2 -29225.532} C_VEL
LIN {X 0,Y 48.387,Z 618.908,A -85,B 0,C 180,E1 -29241.649,E2 -29241.649} C_VEL
LIN {X 0,Y 48.363,Z 619.893,A -85,B 0,C 180,E1 -29250,E2 -29250} C_VEL
LIN {X 0,Y 49.283,Z 620.794,A -85,B 0,C 180,E1 -29266.571,E2 -29266.571} C_VEL
LIN {X 0,Y 53.527,Z 620.374,A -85,B 0,C 180,E1 -29281.68,E2 -29281.68} C_VEL
LIN {X 0,Y 60.822,Z 618.645,A -85,B 0,C 180,E1 -29293.891,E2 -29293.891} C_VEL
LIN {X 0,Y 70.162,Z 615.567,A -85,B 0,C 180,E1 -29303.257,E2 -29303.257} C_VEL
LIN {X 0,Y 80.95,Z 611.059,A -85,B 0,C 180,E1 -29310.246,E2 -29310.246} C_VEL
LIN {X 0,Y 89.687,Z 606.612,A -85,B 0,C 180,E1 -29314.307,E2 -29314.307} C_VEL
LIN {X 0,Y 100.382,Z 600.215,A -85,B 0,C 180,E1 -29318.07,E2 -29318.07} C_VEL
LIN {X 0,Y 111.415,Z 592.285,A -85,B 0,C 180,E1 -29321.114,E2 -29321.114} C_VEL
LIN {X 0,Y 120.748,Z 584.31,A -85,B 0,C 180,E1 -29323.221,E2 -29323.221} C_VEL
LIN {X 0,Y 130.893,Z 574.07,A -85,B 0,C 180,E1 -29325.115,E2 -29325.115} C_VEL
LIN {X 0,Y 140.017,Z 563.027,A -85,B 0,C 180,E1 -29326.527,E2 -29326.527} C_VEL
LIN {X 0,Y 148.411,Z 550.686,A -85,B 0,C 180,E1 -29327.599,E2 -29327.599} C_VEL
LIN {X 0,Y 155.156,Z 538.474,A -85,B 0,C 180,E1 -29328.38,E2 -29328.38} C_VEL
LIN {X 0,Y 160.417,Z 526.677,A -85,B 0,C 180,E1 -29328.933,E2 -29328.933} C_VEL
LIN {X 0,Y 165.282,Z 512.317,A -85,B 0,C 180,E1 -29329.436,E2 -29329.436} C_VEL
LIN {X 0,Y 168.467,Z 498.894,A -85,B 0,C 180,E1 -29329.825,E2 -29329.825} C_VEL
LIN {X 0,Y 168.062,Z 496.991,A -85,B 0,C 180,E1 -29332.19,E2 -29332.19} C_VEL
LIN {X 0,Y 167.885,Z 494.37,A -85,B 0,C 180,E1 -29336.854,E2 -29336.854} C_VEL
LIN {X 0,Y 167.873,Z 494.624,A -85,B 0,C 180,E1 -29338.582,E2 -29338.582} C_VEL
LIN {X 0,Y 168.009,Z 496.589,A -85,B 0,C 180,E1 -29341.96,E2 -29341.96} C_VEL
LIN {X 0,Y 167.962,Z 497.77,A -85,B 0,C 180,E1 -29342.628,E2 -29342.628} C_VEL
LIN {X 0,Y 167.682,Z 499.792,A -85,B 0,C 180,E1 -29343.057,E2 -29343.057} C_VEL
LIN {X 0,Y 166.891,Z 503.538,A -85,B 0,C 180,E1 -29343.32,E2 -29343.32} C_VEL
LIN {X 0,Y 165.725,Z 507.916,A -85,B 0,C 180,E1 -29343.15,E2 -29343.15} C_VEL
LIN {X 0,Y 163.29,Z 515.614,A -85,B 0,C 180,E1 -29342.76,E2 -29342.76} C_VEL
LIN {X 0,Y 162.787,Z 517.1,A -85,B 0,C 180,E1 -29342.791,E2 -29342.791} C_VEL
LIN {X 0,Y 157.524,Z 530.758,A -85,B 0,C 180,E1 -29343.396,E2 -29343.396} C_VEL
LIN {X 0,Y 151.474,Z 542.915,A -85,B 0,C 180,E1 -29344.04,E2 -29344.04} C_VEL
LIN {X 0,Y 144.583,Z 554.163,A -85,B 0,C 180,E1 -29344.826,E2 -29344.826} C_VEL
LIN {X 0,Y 136.166,Z 565.528,A -85,B 0,C 180,E1 -29345.926,E2 -29345.926} C_VEL
LIN {X 0,Y 127.512,Z 575.268,A -85,B 0,C 180,E1 -29347.222,E2 -29347.222} C_VEL
LIN {X 0,Y 117.383,Z 584.829,A -85,B 0,C 180,E1 -29348.936,E2 -29348.936} C_VEL
LIN {X 0,Y 105.872,Z 593.865,A -85,B 0,C 180,E1 -29351.488,E2 -29351.488} C_VEL
LIN {X 0,Y 94.445,Z 601.216,A -85,B 0,C 180,E1 -29354.68,E2 -29354.68} C_VEL
LIN {X 0,Y 81.911,Z 607.739,A -85,B 0,C 180,E1 -29359.303,E2 -29359.303} C_VEL
LIN {X 0,Y 70.037,Z 612.596,A -85,B 0,C 180,E1 -29365.431,E2 -29365.431} C_VEL
LIN {X 0,Y 59.272,Z 615.934,A -85,B 0,C 180,E1 -29373.903,E2 -29373.903} C_VEL
LIN {X 0,Y 50.25,Z 617.854,A -85,B 0,C 180,E1 -29385.63,E2 -29385.63} C_VEL
LIN {X 0,Y 43.769,Z 618.414,A -85,B 0,C 180,E1 -29401.203,E2 -29401.203} C_VEL
LIN {X 0,Y 41.147,Z 617.635,A -85,B 0,C 180,E1 -29420.166,E2 -29420.166} C_VEL
LIN {X 0,Y 41.33,Z 616.751,A -85,B 0,C 180,E1 -29430,E2 -29430} C_VEL
LIN {X 0,Y 42.363,Z 615.539,A -85,B 0,C 180,E1 -29439.549,E2 -29439.549} C_VEL
LIN {X 0,Y 46.973,Z 612.092,A -85,B 0,C 180,E1 -29456.669,E2 -29456.669} C_VEL
LIN {X 0,Y 54.583,Z 607.173,A -85,B 0,C 180,E1 -29470.073,E2 -29470.073} C_VEL
LIN {X 0,Y 61.833,Z 602.409,A -85,B 0,C 180,E1 -29477.627,E2 -29477.627} C_VEL
LIN {X 0,Y 71.135,Z 595.541,A -85,B 0,C 180,E1 -29484.593,E2 -29484.593} C_VEL
LIN {X 0,Y 79.693,Z 588.377,A -85,B 0,C 180,E1 -29489.296,E2 -29489.296} C_VEL
LIN {X 0,Y 88.723,Z 579.751,A -85,B 0,C 180,E1 -29493.014,E2 -29493.014} C_VEL
LIN {X 0,Y 98.048,Z 569.297,A -85,B 0,C 180,E1 -29496.047,E2 -29496.047} C_VEL
LIN {X 0,Y 105.131,Z 559.944,A -85,B 0,C 180,E1 -29498.051,E2 -29498.051} C_VEL
LIN {X 0,Y 112.322,Z 548.727,A -85,B 0,C 180,E1 -29499.805,E2 -29499.805} C_VEL
LIN {X 0,Y 118.813,Z 536.469,A -85,B 0,C 180,E1 -29501.156,E2 -29501.156} C_VEL
LIN {X 0,Y 124.551,Z 522.814,A -85,B 0,C 180,E1 -29502.209,E2 -29502.209} C_VEL
LIN {X 0,Y 128.897,Z 508.898,A -85,B 0,C 180,E1 -29503.037,E2 -29503.037} C_VEL
LIN {X 0,Y 132.056,Z 494.184,A -85,B 0,C 180,E1 -29503.605,E2 -29503.605} C_VEL
LIN {X 0,Y 134.393,Z 475.197,A -85,B 0,C 180,E1 -29504.127,E2 -29504.127} C_VEL
LIN {X 0,Y 133.226,Z 471.384,A -85,B 0,C 180,E1 -29507.817,E2 -29507.817} C_VEL
LIN {X 0,Y 132.468,Z 468.702,A -85,B 0,C 180,E1 -29511.61,E2 -29511.61} C_VEL
LIN {X 0,Y 132.135,Z 467.028,A -85,B 0,C 180,E1 -29516.95,E2 -29516.95} C_VEL
LIN {X 0,Y 132.575,Z 468.967,A -85,B 0,C 180,E1 -29522.658,E2 -29522.658} C_VEL
LIN {X 0,Y 133.495,Z 472.271,A -85,B 0,C 180,E1 -29526.802,E2 -29526.802} C_VEL
LIN {X 0,Y 134.429,Z 475.227,A -85,B 0,C 180,E1 -29529.584,E2 -29529.584} C_VEL
LIN {X 0,Y 131.707,Z 496.776,A -85,B 0,C 180,E1 -29530.109,E2 -29530.109} C_VEL
LIN {X 0,Y 128.403,Z 511.648,A -85,B 0,C 180,E1 -29530.649,E2 -29530.649} C_VEL
LIN {X 0,Y 124.099,Z 525.045,A -85,B 0,C 180,E1 -29531.358,E2 -29531.358} C_VEL
LIN {X 0,Y 118.652,Z 537.853,A -85,B 0,C 180,E1 -29532.233,E2 -29532.233} C_VEL
LIN {X 0,Y 112.012,Z 550.342,A -85,B 0,C 180,E1 -29533.47,E2 -29533.47} C_VEL
LIN {X 0,Y 104.622,Z 561.758,A -85,B 0,C 180,E1 -29535.068,E2 -29535.068} C_VEL
LIN {X 0,Y 95.81,Z 573.244,A -85,B 0,C 180,E1 -29537.529,E2 -29537.529} C_VEL
LIN {X 0,Y 86.327,Z 583.454,A -85,B 0,C 180,E1 -29540.578,E2 -29540.578} C_VEL
LIN {X 0,Y 77.151,Z 591.923,A -85,B 0,C 180,E1 -29544.368,E2 -29544.368} C_VEL
LIN {X 0,Y 67.124,Z 600.023,A -85,B 0,C 180,E1 -29550.258,E2 -29550.258} C_VEL
LIN {X 0,Y 57.811,Z 606.634,A -85,B 0,C 180,E1 -29558.136,E2 -29558.136} C_VEL
LIN {X 0,Y 49.276,Z 612.311,A -85,B 0,C 180,E1 -29570.074,E2 -29570.074} C_VEL
LIN {X 0,Y 44.493,Z 615.588,A -85,B 0,C 180,E1 -29581.715,E2 -29581.715} C_VEL
LIN {X 0,Y 41.367,Z 618.648,A -85,B 0,C 180,E1 -29600.219,E2 -29600.219} C_VEL
LIN {X 0,Y 41.274,Z 619.65,A -85,B 0,C 180,E1 -29610,E2 -29610} C_VEL
LIN {X 0,Y 42.507,Z 620.584,A -85,B 0,C 180,E1 -29629.309,E2 -29629.309} C_VEL
LIN {X 0,Y 47.592,Z 620.196,A -85,B 0,C 180,E1 -29646.205,E2 -29646.205} C_VEL
LIN {X 0,Y 55.887,Z 618.5,A -85,B 0,C 180,E1 -29658.981,E2 -29658.981} C_VEL
LIN {X 0,Y 66.134,Z 615.457,A -85,B 0,C 180,E1 -29668.225,E2 -29668.225} C_VEL
LIN {X 0,Y 77.661,Z 610.985,A -85,B 0,C 180,E1 -29674.815,E2 -29674.815} C_VEL
LIN {X 0,Y 89.953,Z 604.935,A -85,B 0,C 180,E1 -29679.641,E2 -29679.641} C_VEL
LIN {X 0,Y 101.178,Z 598.162,A -85,B 0,C 180,E1 -29682.759,E2 -29682.759} C_VEL
LIN {X 0,Y 112.091,Z 590.205,A -85,B 0,C 180,E1 -29685.178,E2 -29685.178} C_VEL
LIN {X 0,Y 122.547,Z 581.036,A -85,B 0,C 180,E1 -29687.14,E2 -29687.14} C_VEL
LIN {X 0,Y 132.631,Z 570.473,A -85,B 0,C 180,E1 -29688.599,E2 -29688.599} C_VEL
LIN {X 0,Y 141.079,Z 559.835,A -85,B 0,C 180,E1 -29689.687,E2 -29689.687} C_VEL
LIN {X 0,Y 148.755,Z 548.232,A -85,B 0,C 180,E1 -29690.478,E2 -29690.478} C_VEL
LIN {X 0,Y 155.595,Z 535.483,A -85,B 0,C 180,E1 -29691.128,E2 -29691.128} C_VEL
LIN {X 0,Y 161.029,Z 522.634,A -85,B 0,C 180,E1 -29691.594,E2 -29691.594} C_VEL
LIN {X 0,Y 165.538,Z 508.403,A -85,B 0,C 180,E1 -29691.988,E2 -29691.988} C_VEL
LIN {X 0,Y 166.581,Z 504.018,A -85,B 0,C 180,E1 -29692.141,E2 -29692.141} C_VEL
LIN {X 0,Y 166.516,Z 501.337,A -85,B 0,C 180,E1 -29696.977,E2 -29696.977} C_VEL
LIN {X 0,Y 166.484,Z 501.514,A -85,B 0,C 180,E1 -29698.186,E2 -29698.186} C_VEL
LIN {X 0,Y 166.517,Z 503.888,A -85,B 0,C 180,E1 -29702.316,E2 -29702.316} C_VEL
LIN {X 0,Y 162.787,Z 517.1,A -85,B 0,C 180,E1 -29702.791,E2 -29702.791} C_VEL
LIN {X 0,Y 160.777,Z 522.67,A -85,B 0,C 180,E1 -29702.791,E2 -29702.791} C_VEL
LIN {X 0,Y 156.853,Z 531.586,A -85,B 0,C 180,E1 -29702.149,E2 -29702.149} C_VEL
LIN {X 0,Y 152.38,Z 540.289,A -85,B 0,C 180,E1 -29701.482,E2 -29701.482} C_VEL
LIN {X 0,Y 149.473,Z 545.397,A -85,B 0,C 180,E1 -29701.477,E2 -29701.477} C_VEL
LIN {X 0,Y 141.545,Z 557.57,A -85,B 0,C 180,E1 -29702.263,E2 -29702.263} C_VEL
LIN {X 0,Y 133.723,Z 567.54,A -85,B 0,C 180,E1 -29703.091,E2 -29703.091} C_VEL
LIN {X 0,Y 125.082,Z 576.86,A -85,B 0,C 180,E1 -29704.218,E2 -29704.218} C_VEL
LIN {X 0,Y 114.774,Z 586.158,A -85,B 0,C 180,E1 -29705.724,E2 -29705.724} C_VEL
LIN {X 0,Y 103.809,Z 594.402,A -85,B 0,C 180,E1 -29707.783,E2 -29707.783} C_VEL
LIN {X 0,Y 92.876,Z 601.226,A -85,B 0,C 180,E1 -29710.363,E2 -29710.363} C_VEL
LIN {X 0,Y 79.816,Z 607.79,A -85,B 0,C 180,E1 -29714.406,E2 -29714.406} C_VEL
LIN {X 0,Y 67.251,Z 612.686,A -85,B 0,C 180,E1 -29719.862,E2 -29719.862} C_VEL
LIN {X 0,Y 55.556,Z 616.061,A -85,B 0,C 180,E1 -29727.688,E2 -29727.688} C_VEL
LIN {X 0,Y 45.373,Z 618.022,A -85,B 0,C 180,E1 -29739.245,E2 -29739.245} C_VEL
LIN {X 0,Y 37.629,Z 618.624,A -85,B 0,C 180,E1 -29755.924,E2 -29755.924} C_VEL
LIN {X 0,Y 34.122,Z 617.881,A -85,B 0,C 180,E1 -29778.114,E2 -29778.114} C_VEL
LIN {X 0,Y 34.188,Z 617.014,A -85,B 0,C 180,E1 -29790,E2 -29790} C_VEL
LIN {X 0,Y 35.386,Z 615.817,A -85,B 0,C 180,E1 -29801.455,E2 -29801.455} C_VEL
LIN {X 0,Y 40.771,Z 612.405,A -85,B 0,C 180,E1 -29821.139,E2 -29821.139} C_VEL
LIN {X 0,Y 49.388,Z 607.524,A -85,B 0,C 180,E1 -29835.356,E2 -29835.356} C_VEL
LIN {X 0,Y 57.299,Z 602.801,A -85,B 0,C 180,E1 -29842.867,E2 -29842.867} C_VEL
LIN {X 0,Y 67.289,Z 595.977,A -85,B 0,C 180,E1 -29849.502,E2 -29849.502} C_VEL
LIN {X 0,Y 76.332,Z 588.863,A -85,B 0,C 180,E1 -29853.854,E2 -29853.854} C_VEL
LIN {X 0,Y 85.75,Z 580.295,A -85,B 0,C 180,E1 -29857.222,E2 -29857.222} C_VEL
LIN {X 0,Y 95.404,Z 569.909,A -85,B 0,C 180,E1 -29859.92,E2 -29859.92} C_VEL
LIN {X 0,Y 102.701,Z 560.641,A -85,B 0,C 180,E1 -29861.707,E2 -29861.707} C_VEL
LIN {X 0,Y 110.908,Z 548.115,A -85,B 0,C 180,E1 -29863.418,E2 -29863.418} C_VEL
LIN {X 0,Y 116.723,Z 537.417,A -85,B 0,C 180,E1 -29864.44,E2 -29864.44} C_VEL
LIN {X 0,Y 122.586,Z 523.965,A -85,B 0,C 180,E1 -29865.337,E2 -29865.337} C_VEL
LIN {X 0,Y 127.137,Z 509.955,A -85,B 0,C 180,E1 -29866.102,E2 -29866.102} C_VEL
LIN {X 0,Y 130.329,Z 495.871,A -85,B 0,C 180,E1 -29866.581,E2 -29866.581} C_VEL
LIN {X 0,Y 132.5,Z 479.625,A -85,B 0,C 180,E1 -29867.026,E2 -29867.026} C_VEL
LIN {X 0,Y 131.735,Z 476.908,A -85,B 0,C 180,E1 -29870.402,E2 -29870.402} C_VEL
LIN {X 0,Y 131.428,Z 475.482,A -85,B 0,C 180,E1 -29872.703,E2 -29872.703} C_VEL
LIN {X 0,Y 131.266,Z 474.087,A -85,B 0,C 180,E1 -29876.93,E2 -29876.93} C_VEL
LIN {X 0,Y 131.594,Z 475.906,A -85,B 0,C 180,E1 -29882.103,E2 -29882.103} C_VEL
LIN {X 0,Y 132.313,Z 478.963,A -85,B 0,C 180,E1 -29885.906,E2 -29885.906} C_VEL
LIN {X 0,Y 132.51,Z 479.697,A -85,B 0,C 180,E1 -29886.657,E2 -29886.657} C_VEL
LIN {X 0,Y 130.483,Z 495.542,A -85,B 0,C 180,E1 -29887.05,E2 -29887.05} C_VEL
LIN {X 0,Y 127.405,Z 509.726,A -85,B 0,C 180,E1 -29887.479,E2 -29887.479} C_VEL
LIN {X 0,Y 123.201,Z 523.057,A -85,B 0,C 180,E1 -29888.033,E2 -29888.033} C_VEL
LIN {X 0,Y 118.205,Z 535.144,A -85,B 0,C 180,E1 -29888.726,E2 -29888.726} C_VEL
LIN {X 0,Y 111.419,Z 548.113,A -85,B 0,C 180,E1 -29889.751,E2 -29889.751} C_VEL
LIN {X 0,Y 103.835,Z 559.883,A -85,B 0,C 180,E1 -29891.071,E2 -29891.071} C_VEL
LIN {X 0,Y 95.889,Z 570.271,A -85,B 0,C 180,E1 -29892.875,E2 -29892.875} C_VEL
LIN {X 0,Y 87.319,Z 579.693,A -85,B 0,C 180,E1 -29895.027,E2 -29895.027} C_VEL
LIN {X 0,Y 77.638,Z 588.761,A -85,B 0,C 180,E1 -29898.11,E2 -29898.11} C_VEL
LIN {X 0,Y 66.786,Z 597.444,A -85,B 0,C 180,E1 -29902.965,E2 -29902.965} C_VEL
LIN {X 0,Y 55.557,Z 605.104,A -85,B 0,C 180,E1 -29910.395,E2 -29910.395} C_VEL
LIN {X 0,Y 46.282,Z 610.715,A -85,B 0,C 180,E1 -29920.604,E2 -29920.604} C_VEL
LIN {X 0,Y 38.331,Z 615.291,A -85,B 0,C 180,E1 -29936.63,E2 -29936.63} C_VEL
LIN {X 0,Y 34.366,Z 618.388,A -85,B 0,C 180,E1 -29958.2,E2 -29958.2} C_VEL
LIN {X 0,Y 34.158,Z 619.407,A -85,B 0,C 180,E1 -29970,E2 -29970} C_VEL
LIN {X 0,Y 35.845,Z 620.373,A -85,B 0,C 180,E1 -29993.087,E2 -29993.087} C_VEL
LIN {X 0,Y 42.039,Z 620.018,A -85,B 0,C 180,E1 -30011.967,E2 -30011.967} C_VEL
LIN {X 0,Y 51.48,Z 618.356,A -85,B 0,C 180,E1 -30024.994,E2 -30024.994} C_VEL
LIN {X 0,Y 62.673,Z 615.347,A -85,B 0,C 180,E1 -30033.777,E2 -30033.777} C_VEL
LIN {X 0,Y 74.9,Z 610.912,A -85,B 0,C 180,E1 -30039.767,E2 -30039.767} C_VEL
LIN {X 0,Y 87.727,Z 604.915,A -85,B 0,C 180,E1 -30044.012,E2 -30044.012} C_VEL
LIN {X 0,Y 99.304,Z 598.19,A -85,B 0,C 180,E1 -30046.68,E2 -30046.68} C_VEL
LIN {X 0,Y 109.865,Z 590.775,A -85,B 0,C 180,E1 -30048.636,E2 -30048.636} C_VEL
LIN {X 0,Y 121.163,Z 581.171,A -85,B 0,C 180,E1 -30050.418,E2 -30050.418} C_VEL
LIN {X 0,Y 131.415,Z 570.675,A -85,B 0,C 180,E1 -30051.627,E2 -30051.627} C_VEL
LIN {X 0,Y 139.984,Z 560.118,A -85,B 0,C 180,E1 -30052.541,E2 -30052.541} C_VEL
LIN {X 0,Y 147.75,Z 548.62,A -85,B 0,C 180,E1 -30053.184,E2 -30053.184} C_VEL
LIN {X 0,Y 154.662,Z 536.012,A -85,B 0,C 180,E1 -30053.718,E2 -30053.718} C_VEL
LIN {X 0,Y 160.148,Z 523.365,A -85,B 0,C 180,E1 -30054.097,E2 -30054.097} C_VEL
LIN {X 0,Y 164.593,Z 509.831,A -85,B 0,C 180,E1 -30054.433,E2 -30054.433} C_VEL
LIN {X 0,Y 164.831,Z 508.173,A -85,B 0,C 180,E1 -30057.557,E2 -30057.557} C_VEL
LIN {X 0,Y 164.606,Z 509.521,A -85,B 0,C 180,E1 -30060.001,E2 -30060.001} C_VEL
LIN {X 0,Y 160.534,Z 522.067,A -85,B 0,C 180,E1 -30060.451,E2 -30060.451} C_VEL
LIN {X 0,Y 155.381,Z 534.223,A -85,B 0,C 180,E1 -30060.944,E2 -30060.944} C_VEL
LIN {X 0,Y 149.473,Z 545.397,A -85,B 0,C 180,E1 -30061.477,E2 -30061.477} C_VEL
LIN {X 0,Y 147.398,Z 548.812,A -85,B 0,C 180,E1 -30061.393,E2 -30061.393} C_VEL
LIN {X 0,Y 139.998,Z 559.339,A -85,B 0,C 180,E1 -30059.747,E2 -30059.747} C_VEL
LIN {X 0,Y 137.531,Z 562.454,A -85,B 0,C 180,E1 -30059.687,E2 -30059.687} C_VEL
LIN {X 0,Y 129.751,Z 571.552,A -85,B 0,C 180,E1 -30060.409,E2 -30060.409} C_VEL
LIN {X 0,Y 119.512,Z 581.608,A -85,B 0,C 180,E1 -30061.478,E2 -30061.478} C_VEL
LIN {X 0,Y 109.067,Z 590.136,A -85,B 0,C 180,E1 -30062.861,E2 -30062.861} C_VEL
LIN {X 0,Y 96.987,Z 598.249,A -85,B 0,C 180,E1 -30064.9,E2 -30064.9} C_VEL
LIN {X 0,Y 85.056,Z 604.759,A -85,B 0,C 180,E1 -30067.472,E2 -30067.472} C_VEL
LIN {X 0,Y 71.678,Z 610.507,A -85,B 0,C 180,E1 -30071.343,E2 -30071.343} C_VEL
LIN {X 0,Y 58.759,Z 614.665,A -85,B 0,C 180,E1 -30076.896,E2 -30076.896} C_VEL
LIN {X 0,Y 46.682,Z 617.359,A -85,B 0,C 180,E1 -30085.407,E2 -30085.407} C_VEL
LIN {X 0,Y 36.18,Z 618.675,A -85,B 0,C 180,E1 -30099.015,E2 -30099.015} C_VEL
LIN {X 0,Y 28.835,Z 618.644,A -85,B 0,C 180,E1 -30120.826,E2 -30120.826} C_VEL
LIN {X 0,Y 27.051,Z 617.276,A -85,B 0,C 180,E1 -30150,E2 -30150} C_VEL
LIN {X 0,Y 28.457,Z 616.096,A -85,B 0,C 180,E1 -30164.297,E2 -30164.297} C_VEL
LIN {X 0,Y 34.894,Z 612.719,A -85,B 0,C 180,E1 -30187.171,E2 -30187.171} C_VEL
LIN {X 0,Y 44.703,Z 607.875,A -85,B 0,C 180,E1 -30201.818,E2 -30201.818} C_VEL
LIN {X 0,Y 53.331,Z 603.193,A -85,B 0,C 180,E1 -30208.93,E2 -30208.93} C_VEL
LIN {X 0,Y 63.996,Z 596.413,A -85,B 0,C 180,E1 -30214.957,E2 -30214.957} C_VEL
LIN {X 0,Y 73.487,Z 589.351,A -85,B 0,C 180,E1 -30218.815,E2 -30218.815} C_VEL
LIN {X 0,Y 83.272,Z 580.839,A -85,B 0,C 180,E1 -30221.704,E2 -30221.704} C_VEL
LIN {X 0,Y 93.219,Z 570.52,A -85,B 0,C 180,E1 -30223.993,E2 -30223.993} C_VEL
LIN {X 0,Y 100.708,Z 561.329,A -85,B 0,C 180,E1 -30225.523,E2 -30225.523} C_VEL
LIN {X 0,Y 109.105,Z 548.917,A -85,B 0,C 180,E1 -30226.969,E2 -30226.969} C_VEL
LIN {X 0,Y 115.884,Z 536.606,A -85,B 0,C 180,E1 -30227.933,E2 -30227.933} C_VEL
LIN {X 0,Y 121.836,Z 522.881,A -85,B 0,C 180,E1 -30228.695,E2 -30228.695} C_VEL
LIN {X 0,Y 126.336,Z 508.943,A -85,B 0,C 180,E1 -30229.3,E2 -30229.3} C_VEL
LIN {X 0,Y 129.601,Z 494.123,A -85,B 0,C 180,E1 -30229.728,E2 -30229.728} C_VEL
LIN {X 0,Y 130.901,Z 484.522,A -85,B 0,C 180,E1 -30229.992,E2 -30229.992} C_VEL
LIN {X 0,Y 130.47,Z 482.329,A -85,B 0,C 180,E1 -30233.477,E2 -30233.477} C_VEL
LIN {X 0,Y 130.387,Z 481.267,A -85,B 0,C 180,E1 -30237.296,E2 -30237.296} C_VEL
LIN {X 0,Y 130.602,Z 482.751,A -85,B 0,C 180,E1 -30241.348,E2 -30241.348} C_VEL
LIN {X 0,Y 130.937,Z 484.469,A -85,B 0,C 180,E1 -30243.753,E2 -30243.753} C_VEL
LIN {X 0,Y 128.537,Z 500.111,A -85,B 0,C 180,E1 -30244.035,E2 -30244.035} C_VEL
LIN {X 0,Y 124.887,Z 514.547,A -85,B 0,C 180,E1 -30244.457,E2 -30244.457} C_VEL
LIN {X 0,Y 119.931,Z 528.302,A -85,B 0,C 180,E1 -30245.013,E2 -30245.013} C_VEL
LIN {X 0,Y 113.879,Z 541.135,A -85,B 0,C 180,E1 -30245.665,E2 -30245.665} C_VEL
LIN {X 0,Y 106.988,Z 552.898,A -85,B 0,C 180,E1 -30246.523,E2 -30246.523} C_VEL
LIN {X 0,Y 99.288,Z 563.8,A -85,B 0,C 180,E1 -30247.718,E2 -30247.718} C_VEL
LIN {X 0,Y 90.822,Z 573.903,A -85,B 0,C 180,E1 -30249.395,E2 -30249.395} C_VEL
LIN {X 0,Y 80.723,Z 583.93,A -85,B 0,C 180,E1 -30251.642,E2 -30251.642} C_VEL
LIN {X 0,Y 70.787,Z 592.248,A -85,B 0,C 180,E1 -30254.537,E2 -30254.537} C_VEL
LIN {X 0,Y 59.593,Z 600.216,A -85,B 0,C 180,E1 -30259.364,E2 -30259.364} C_VEL
LIN {X 0,Y 50.177,Z 605.909,A -85,B 0,C 180,E1 -30265.133,E2 -30265.133} C_VEL
LIN {X 0,Y 39.375,Z 611.646,A -85,B 0,C 180,E1 -30276.566,E2 -30276.566} C_VEL
LIN {X 0,Y 32.587,Z 614.995,A -85,B 0,C 180,E1 -30289.685,E2 -30289.685} C_VEL
LIN {X 0,Y 27.418,Z 618.127,A -85,B 0,C 180,E1 -30315.148,E2 -30315.148} C_VEL
LIN {X 0,Y 27.048,Z 619.163,A -85,B 0,C 180,E1 -30330,E2 -30330} C_VEL
LIN {X 0,Y 29.418,Z 620.162,A -85,B 0,C 180,E1 -30358.541,E2 -30358.541} C_VEL
LIN {X 0,Y 37.04,Z 619.84,A -85,B 0,C 180,E1 -30379.371,E2 -30379.371} C_VEL
LIN {X 0,Y 47.741,Z 618.211,A -85,B 0,C 180,E1 -30392.036,E2 -30392.036} C_VEL
LIN {X 0,Y 59.858,Z 615.237,A -85,B 0,C 180,E1 -30399.927,E2 -30399.927} C_VEL
LIN {X 0,Y 72.743,Z 610.838,A -85,B 0,C 180,E1 -30405.042,E2 -30405.042} C_VEL
LIN {X 0,Y 86.038,Z 604.887,A -85,B 0,C 180,E1 -30408.578,E2 -30408.578} C_VEL
LIN {X 0,Y 97.911,Z 598.211,A -85,B 0,C 180,E1 -30410.732,E2 -30410.732} C_VEL
LIN {X 0,Y 108.366,Z 591.068,A -85,B 0,C 180,E1 -30412.266,E2 -30412.266} C_VEL
LIN {X 0,Y 118.461,Z 582.847,A -85,B 0,C 180,E1 -30413.571,E2 -30413.571} C_VEL
LIN {X 0,Y 128.838,Z 572.79,A -85,B 0,C 180,E1 -30414.56,E2 -30414.56} C_VEL
LIN {X 0,Y 138.373,Z 561.572,A -85,B 0,C 180,E1 -30415.364,E2 -30415.364} C_VEL
LIN {X 0,Y 147.078,Z 549.006,A -85,B 0,C 180,E1 -30415.919,E2 -30415.919} C_VEL
LIN {X 0,Y 154.048,Z 536.54,A -85,B 0,C 180,E1 -30416.335,E2 -30416.335} C_VEL
LIN {X 0,Y 160.015,Z 522.964,A -85,B 0,C 180,E1 -30416.645,E2 -30416.645} C_VEL
LIN {X 0,Y 162.336,Z 516.455,A -85,B 0,C 180,E1 -30416.767,E2 -30416.767} C_VEL
LIN {X 0,Y 162.712,Z 515.322,A -85,B 0,C 180,E1 -30416.947,E2 -30416.947} C_VEL
LIN {X 0,Y 162.786,Z 515.073,A -85,B 0,C 180,E1 -30417.526,E2 -30417.526} C_VEL
LIN {X 0,Y 162.435,Z 516.113,A -85,B 0,C 180,E1 -30417.752,E2 -30417.752} C_VEL
LIN {X 0,Y 157.419,Z 529.247,A -85,B 0,C 180,E1 -30418.175,E2 -30418.175} C_VEL
LIN {X 0,Y 151.142,Z 541.963,A -85,B 0,C 180,E1 -30418.613,E2 -30418.613} C_VEL
LIN {X 0,Y 143.205,Z 554.761,A -85,B 0,C 180,E1 -30419.207,E2 -30419.207} C_VEL
LIN {X 0,Y 137.531,Z 562.454,A -85,B 0,C 180,E1 -30419.687,E2 -30419.687} C_VEL
LIN {X 0,Y 133.747,Z 567.056,A -85,B 0,C 180,E1 -30419.75,E2 -30419.75} C_VEL
LIN {X 0,Y 127.05,Z 574.275,A -85,B 0,C 180,E1 -30419.052,E2 -30419.052} C_VEL
LIN {X 0,Y 120.011,Z 581.039,A -85,B 0,C 180,E1 -30418.312,E2 -30418.312} C_VEL
LIN {X 0,Y 115.58,Z 584.842,A -85,B 0,C 180,E1 -30418.385,E2 -30418.385} C_VEL
LIN {X 0,Y 105.421,Z 592.55,A -85,B 0,C 180,E1 -30419.478,E2 -30419.478} C_VEL
LIN {X 0,Y 93.137,Z 600.256,A -85,B 0,C 180,E1 -30421.156,E2 -30421.156} C_VEL
LIN {X 0,Y 80.952,Z 606.403,A -85,B 0,C 180,E1 -30423.274,E2 -30423.274} C_VEL
LIN {X 0,Y 69.966,Z 610.813,A -85,B 0,C 180,E1 -30425.767,E2 -30425.767} C_VEL
LIN {X 0,Y 57.078,Z 614.774,A -85,B 0,C 180,E1 -30429.932,E2 -30429.932} C_VEL
LIN {X 0,Y 44.067,Z 617.503,A -85,B 0,C 180,E1 -30436.887,E2 -30436.887} C_VEL
LIN {X 0,Y 32.133,Z 618.854,A -85,B 0,C 180,E1 -30448.972,E2 -30448.972} C_VEL
LIN {X 0,Y 22.836,Z 618.864,A -85,B 0,C 180,E1 -30472.01,E2 -30472.01} C_VEL
LIN {X 0,Y 19.93,Z 617.537,A -85,B 0,C 180,E1 -30510,E2 -30510} C_VEL
LIN {X 0,Y 21.641,Z 616.375,A -85,B 0,C 180,E1 -30528.95,E2 -30528.95} C_VEL
LIN {X 0,Y 29.563,Z 613.033,A -85,B 0,C 180,E1 -30555.492,E2 -30555.492} C_VEL
LIN {X 0,Y 40.705,Z 608.227,A -85,B 0,C 180,E1 -30569.684,E2 -30569.684} C_VEL
LIN {X 0,Y 50.044,Z 603.586,A -85,B 0,C 180,E1 -30575.895,E2 -30575.895} C_VEL
LIN {X 0,Y 61.337,Z 596.85,A -85,B 0,C 180,E1 -30580.954,E2 -30580.954} C_VEL
LIN {X 0,Y 71.238,Z 589.831,A -85,B 0,C 180,E1 -30584.125,E2 -30584.125} C_VEL
LIN {X 0,Y 81.333,Z 581.372,A -85,B 0,C 180,E1 -30586.429,E2 -30586.429} C_VEL
LIN {X 0,Y 91.521,Z 571.134,A -85,B 0,C 180,E1 -30588.252,E2 -30588.252} C_VEL
LIN {X 0,Y 100.029,Z 560.871,A -85,B 0,C 180,E1 -30589.61,E2 -30589.61} C_VEL
LIN {X 0,Y 107.735,Z 549.719,A -85,B 0,C 180,E1 -30590.623,E2 -30590.623} C_VEL
LIN {X 0,Y 114.614,Z 537.555,A -85,B 0,C 180,E1 -30591.391,E2 -30591.391} C_VEL
LIN {X 0,Y 120.654,Z 524.035,A -85,B 0,C 180,E1 -30591.976,E2 -30591.976} C_VEL
LIN {X 0,Y 125.464,Z 509.573,A -85,B 0,C 180,E1 -30592.491,E2 -30592.491} C_VEL
LIN {X 0,Y 128.61,Z 495.835,A -85,B 0,C 180,E1 -30592.834,E2 -30592.834} C_VEL
LIN {X 0,Y 129.567,Z 489.737,A -85,B 0,C 180,E1 -30593.019,E2 -30593.019} C_VEL
LIN {X 0,Y 129.5,Z 488.326,A -85,B 0,C 180,E1 -30596.888,E2 -30596.888} C_VEL
LIN {X 0,Y 129.605,Z 489.637,A -85,B 0,C 180,E1 -30600.702,E2 -30600.702} C_VEL
LIN {X 0,Y 126.986,Z 503.877,A -85,B 0,C 180,E1 -30600.98,E2 -30600.98} C_VEL
LIN {X 0,Y 123.057,Z 517.689,A -85,B 0,C 180,E1 -30601.276,E2 -30601.276} C_VEL
LIN {X 0,Y 117.769,Z 531.27,A -85,B 0,C 180,E1 -30601.735,E2 -30601.735} C_VEL
LIN {X 0,Y 111.649,Z 543.455,A -85,B 0,C 180,E1 -30602.21,E2 -30602.21} C_VEL
LIN {X 0,Y 103.801,Z 556.066,A -85,B 0,C 180,E1 -30602.985,E2 -30602.985} C_VEL
LIN {X 0,Y 96.143,Z 566.192,A -85,B 0,C 180,E1 -30603.935,E2 -30603.935} C_VEL
LIN {X 0,Y 86.474,Z 576.921,A -85,B 0,C 180,E1 -30605.396,E2 -30605.396} C_VEL
LIN {X 0,Y 76.16,Z 586.412,A -85,B 0,C 180,E1 -30607.264,E2 -30607.264} C_VEL
LIN {X 0,Y 65.959,Z 594.279,A -85,B 0,C 180,E1 -30609.744,E2 -30609.744} C_VEL
LIN {X 0,Y 54.318,Z 601.826,A -85,B 0,C 180,E1 -30613.982,E2 -30613.982} C_VEL
LIN {X 0,Y 44.652,Z 607.056,A -85,B 0,C 180,E1 -30619.207,E2 -30619.207} C_VEL
LIN {X 0,Y 32.748,Z 612.564,A -85,B 0,C 180,E1 -30630.862,E2 -30630.862} C_VEL
LIN {X 0,Y 23.314,Z 616.462,A -85,B 0,C 180,E1 -30652.924,E2 -30652.924} C_VEL
LIN {X 0,Y 19.951,Z 618.92,A -85,B 0,C 180,E1 -30690,E2 -30690} C_VEL
LIN {X 0,Y 23.41,Z 619.952,A -85,B 0,C 180,E1 -30726.899,E2 -30726.899} C_VEL
LIN {X 0,Y 32.846,Z 619.663,A -85,B 0,C 180,E1 -30748.855,E2 -30748.855} C_VEL
LIN {X 0,Y 44.838,Z 618.067,A -85,B 0,C 180,E1 -30760.124,E2 -30760.124} C_VEL
LIN {X 0,Y 57.799,Z 615.127,A -85,B 0,C 180,E1 -30766.589,E2 -30766.589} C_VEL
LIN {X 0,Y 71.238,Z 610.765,A -85,B 0,C 180,E1 -30770.583,E2 -30770.583} C_VEL
LIN {X 0,Y 84.915,Z 604.853,A -85,B 0,C 180,E1 -30773.29,E2 -30773.29} C_VEL
LIN {X 0,Y 97.018,Z 598.223,A -85,B 0,C 180,E1 -30774.891,E2 -30774.891} C_VEL
LIN {X 0,Y 108.897,Z 590.214,A -85,B 0,C 180,E1 -30776.151,E2 -30776.151} C_VEL
LIN {X 0,Y 119.621,Z 581.441,A -85,B 0,C 180,E1 -30777.143,E2 -30777.143} C_VEL
LIN {X 0,Y 122.838,Z 578.448,A -85,B 0,C 180,E1 -30777.382,E2 -30777.382} C_VEL
LIN {X 0,Y 124.232,Z 577.136,A -85,B 0,C 180,E1 -30777.677,E2 -30777.677} C_VEL
LIN {X 0,Y 115.58,Z 584.842,A -85,B 0,C 180,E1 -30778.385,E2 -30778.385} C_VEL
LIN {X 0,Y 114.868,Z 586.383,A -85,B 0,C 180,E1 -30778.454,E2 -30778.454} C_VEL
LIN {X 0,Y 114.868,Z 615.893,A -85,B 0,C 180,E1 -30778.454,E2 -30778.454} C_VEL
LIN {X 0,Y 86.258,Z 615.893,A -85,B 0,C 180,E1 -30777.803,E2 -30777.803} C_VEL
LIN {X 0,Y 84.26,Z 613.893,A -85,B 0,C 180,E1 -30777.741,E2 -30777.741} C_VEL
LIN {X 0,Y 84.26,Z 607.974,A -85,B 0,C 180,E1 -30777.741,E2 -30777.741} C_VEL
LIN {X 0,Y 81.521,Z 606.133,A -85,B 0,C 180,E1 -30778.075,E2 -30778.075} C_VEL
LIN {X 0,Y 68.678,Z 611.213,A -85,B 0,C 180,E1 -30780.002,E2 -30780.002} C_VEL
LIN {X 0,Y 56.284,Z 614.882,A -85,B 0,C 180,E1 -30782.669,E2 -30782.669} C_VEL
LIN {X 0,Y 42.535,Z 617.647,A -85,B 0,C 180,E1 -30787.54,E2 -30787.54} C_VEL
LIN {X 0,Y 29.327,Z 619.032,A -85,B 0,C 180,E1 -30796.552,E2 -30796.552} C_VEL
LIN {X 0,Y 17.725,Z 619.079,A -85,B 0,C 180,E1 -30817.536,E2 -30817.536} C_VEL
LIN {X 0,Y 12.78,Z 617.794,A -85,B 0,C 180,E1 -30869.999,E2 -30869.999} C_VEL
LIN {X 0,Y 15.092,Z 616.653,A -85,B 0,C 180,E1 -30897.754,E2 -30897.754} C_VEL
LIN {X 0,Y 25.114,Z 613.346,A -85,B 0,C 180,E1 -30927.087,E2 -30927.087} C_VEL
LIN {X 0,Y 37.635,Z 608.578,A -85,B 0,C 180,E1 -30939.016,E2 -30939.016} C_VEL
LIN {X 0,Y 47.597,Z 603.975,A -85,B 0,C 180,E1 -30943.688,E2 -30943.688} C_VEL
LIN {X 0,Y 59.404,Z 597.288,A -85,B 0,C 180,E1 -30947.425,E2 -30947.425} C_VEL
LIN {X 0,Y 69.638,Z 590.301,A -85,B 0,C 180,E1 -30949.725,E2 -30949.725} C_VEL
LIN {X 0,Y 79.973,Z 581.893,A -85,B 0,C 180,E1 -30951.349,E2 -30951.349} C_VEL
LIN {X 0,Y 90.346,Z 571.748,A -85,B 0,C 180,E1 -30952.653,E2 -30952.653} C_VEL
LIN {X 0,Y 99,Z 561.565,A -85,B 0,C 180,E1 -30953.634,E2 -30953.634} C_VEL
LIN {X 0,Y 107.681,Z 549.106,A -85,B 0,C 180,E1 -30954.436,E2 -30954.436} C_VEL
LIN {X 0,Y 114.644,Z 536.745,A -85,B 0,C 180,E1 -30954.964,E2 -30954.964} C_VEL
LIN {X 0,Y 120.583,Z 523.358,A -85,B 0,C 180,E1 -30955.362,E2 -30955.362} C_VEL
LIN {X 0,Y 125.257,Z 509.26,A -85,B 0,C 180,E1 -30955.744,E2 -30955.744} C_VEL
LIN {X 0,Y 128.234,Z 496.341,A -85,B 0,C 180,E1 -30955.989,E2 -30955.989} C_VEL
LIN {X 0,Y 128.374,Z 495.591,A -85,B 0,C 180,E1 -30956.16,E2 -30956.16} C_VEL
LIN {X 0,Y 128.389,Z 495.565,A -85,B 0,C 180,E1 -30957.623,E2 -30957.623} C_VEL
LIN {X 0,Y 124.997,Z 510.233,A -85,B 0,C 180,E1 -30957.883,E2 -30957.883} C_VEL
LIN {X 0,Y 120.455,Z 523.775,A -85,B 0,C 180,E1 -30958.104,E2 -30958.104} C_VEL
LIN {X 0,Y 115.126,Z 535.887,A -85,B 0,C 180,E1 -30958.389,E2 -30958.389} C_VEL
LIN {X 0,Y 108.078,Z 548.591,A -85,B 0,C 180,E1 -30958.745,E2 -30958.745} C_VEL
LIN {X 0,Y 100.155,Z 560.168,A -85,B 0,C 180,E1 -30959.247,E2 -30959.247} C_VEL
LIN {X 0,Y 91.361,Z 570.81,A -85,B 0,C 180,E1 -30960.11,E2 -30960.11} C_VEL
LIN {X 0,Y 80.838,Z 581.356,A -85,B 0,C 180,E1 -30961.233,E2 -30961.233} C_VEL
LIN {X 0,Y 70.349,Z 590.039,A -85,B 0,C 180,E1 -30962.573,E2 -30962.573} C_VEL
LIN {X 0,Y 58.203,Z 598.365,A -85,B 0,C 180,E1 -30965.029,E2 -30965.029} C_VEL
LIN {X 0,Y 45.682,Z 605.299,A -85,B 0,C 180,E1 -30968.847,E2 -30968.847} C_VEL
LIN {X 0,Y 32.918,Z 610.98,A -85,B 0,C 180,E1 -30976.111,E2 -30976.111} C_VEL
LIN {X 0,Y 23.57,Z 614.4,A -85,B 0,C 180,E1 -30986.557,E2 -30986.557} C_VEL
LIN {X 0,Y 14.135,Z 617.606,A -85,B 0,C 180,E1 -31020.185,E2 -31020.185} C_VEL
LIN {X 0,Y 12.842,Z 618.677,A -85,B 0,C 180,E1 -31050.001,E2 -31050.001} C_VEL
LIN {X 0,Y 18.216,Z 619.741,A -85,B 0,C 180,E1 -31100.498,E2 -31100.498} C_VEL
LIN {X 0,Y 29.791,Z 619.485,A -85,B 0,C 180,E1 -31120.671,E2 -31120.671} C_VEL
LIN {X 0,Y 42.939,Z 617.923,A -85,B 0,C 180,E1 -31129.121,E2 -31129.121} C_VEL
LIN {X 0,Y 56.571,Z 615.018,A -85,B 0,C 180,E1 -31133.634,E2 -31133.634} C_VEL
LIN {X 0,Y 70.422,Z 610.691,A -85,B 0,C 180,E1 -31136.333,E2 -31136.333} C_VEL
LIN {X 0,Y 77.391,Z 607.957,A -85,B 0,C 180,E1 -31137.31,E2 -31137.31} C_VEL
LIN {X 0,Y 81.521,Z 606.133,A -85,B 0,C 180,E1 -31138.075,E2 -31138.075} C_VEL
LIN {X 0,Y 84.227,Z 607.972,A -85,B 0,C 180,E1 -31138.534,E2 -31138.534} C_VEL
LIN {X 0,Y 84.227,Z 628.82,A -85,B 0,C 180,E1 -31138.534,E2 -31138.534} C_VEL
LIN {X 0,Y 37.325,Z 628.82,A -85,B 0,C 180,E1 -31134.268,E2 -31134.268} C_VEL
LIN {X 0,Y 35.343,Z 626.82,A -85,B 0,C 180,E1 -31133.837,E2 -31133.837} C_VEL
LIN {X 0,Y 35.343,Z 620.707,A -85,B 0,C 180,E1 -31133.837,E2 -31133.837} C_VEL
LIN {X 0,Y 35.187,Z 618.707,A -85,B 0,C 180,E1 -31137.003,E2 -31137.003} C_VEL
LIN {X 0,Y 35.14,Z 618.67,A -85,B 0,C 180,E1 -31139.678,E2 -31139.678} C_VEL
LIN {X 0,Y 21.22,Z 619.418,A -85,B 0,C 180,E1 -31146.507,E2 -31146.507} C_VEL
LIN {X 0,Y 8.466,Z 618.833,A -85,B 0,C 180,E1 -31173.883,E2 -31173.883} C_VEL
LIN {X 0,Y 5.645,Z 618.044,A -85,B 0,C 180,E1 -31229.999,E2 -31229.999} C_VEL
LIN {X 0,Y 9.412,Z 616.924,A -85,B 0,C 180,E1 -31278.3,E2 -31278.3} C_VEL
LIN {X 0,Y 22.082,Z 613.66,A -85,B 0,C 180,E1 -31302.7,E2 -31302.7} C_VEL
LIN {X 0,Y 35.716,Z 608.93,A -85,B 0,C 180,E1 -31309.684,E2 -31309.684} C_VEL
LIN {X 0,Y 46.364,Z 604.234,A -85,B 0,C 180,E1 -31312.226,E2 -31312.226} C_VEL
LIN {X 0,Y 58.275,Z 597.72,A -85,B 0,C 180,E1 -31314.226,E2 -31314.226} C_VEL
LIN {X 0,Y 70.475,Z 589.467,A -85,B 0,C 180,E1 -31315.711,E2 -31315.711} C_VEL
LIN {X 0,Y 77.461,Z 583.893,A -85,B 0,C 180,E1 -31316.376,E2 -31316.376} C_VEL
LIN {X 0,Y 66.853,Z 592.112,A -85,B 0,C 180,E1 -31317.038,E2 -31317.038} C_VEL
LIN {X 0,Y 54.486,Z 599.993,A -85,B 0,C 180,E1 -31318.422,E2 -31318.422} C_VEL
LIN {X 0,Y 42.168,Z 606.311,A -85,B 0,C 180,E1 -31320.433,E2 -31320.433} C_VEL
LIN {X 0,Y 28.219,Z 611.905,A -85,B 0,C 180,E1 -31325.024,E2 -31325.024} C_VEL
LIN {X 0,Y 14.698,Z 615.903,A -85,B 0,C 180,E1 -31337.009,E2 -31337.009} C_VEL
LIN {X 0,Y 8.696,Z 617.345,A -85,B 0,C 180,E1 -31356.088,E2 -31356.088} C_VEL
LIN {X 0,Y 5.726,Z 618.434,A -85,B 0,C 180,E1 -31410.001,E2 -31410.001} C_VEL
LIN {X 0,Y 8.747,Z 619.15,A -85,B 0,C 180,E1 -31463.462,E2 -31463.462} C_VEL
LIN {X 0,Y 21.383,Z 619.581,A -85,B 0,C 180,E1 -31490.393,E2 -31490.393} C_VEL
LIN {X 0,Y 35.187,Z 618.707,A -85,B 0,C 180,E1 -31497.003,E2 -31497.003} C_VEL
LIN {X 0,Y 35.187,Z 618.707,A -85,B 0,C 180,E1 -31497.003,E2 -31497.003}

QRS_NEXT_CUT()

QRS_NEXT()
QRS_HOME()

END
